ABB RAPID module: CurvedAlign3DP_R7.modx

MODULE CurvedAlign3DP

	VAR jointtarget SDP_0 := [[-4.75, 34.73, 8.1, 0, 47.17, -94.75], [9E9, 9E9, 9E9, 9E9, 9E9, 9E9]];
	VAR jointtarget SDP_1 := [[-3.57, 34.64, 8.25, 0, 47.11, -93.57], [9E9, 9E9, 9E9, 9E9, 9E9, 9E9]];
	VAR jointtarget SDP_2 := [[-2.38, 34.58, 8.36, 0, 47.06, -92.38], [9E9, 9E9, 9E9, 9E9, 9E9, 9E9]];
	VAR jointtarget SDP_3 := [[-1.19, 34.54, 8.43, 0, 47.03, -91.19], [9E9, 9E9, 9E9, 9E9, 9E9, 9E9]];
	VAR jointtarget SDP_4 := [[0, 34.52, 8.45, 0, 47.02, -90], [9E9, 9E9, 9E9, 9E9, 9E9, 9E9]];
	VAR jointtarget SDP_5 := [[1.19, 34.54, 8.43, 0, 47.03, -88.81], [9E9, 9E9, 9E9, 9E9, 9E9, 9E9]];
	VAR jointtarget SDP_6 := [[2.38, 34.58, 8.36, 0, 47.06, -87.62], [9E9, 9E9, 9E9, 9E9, 9E9, 9E9]];
	VAR jointtarget SDP_7 := [[3.57, 34.64, 8.25, 0, 47.11, -86.43], [9E9, 9E9, 9E9, 9E9, 9E9, 9E9]];
	VAR jointtarget SDP_8 := [[4.75, 34.73, 8.1, 0, 47.17, -85.25], [9E9, 9E9, 9E9, 9E9, 9E9, 9E9]];
	VAR jointtarget SDP_9 := [[5.93, 34.85, 7.9, 0, 47.25, -84.07], [9E9, 9E9, 9E9, 9E9, 9E9, 9E9]];
	VAR jointtarget SDP_10 := [[6.27, 34.91, 7.79, 0, 47.3, -79.23], [9E9, 9E9, 9E9, 9E9, 9E9, 9E9]];
	VAR jointtarget SDP_11 := [[6.6, 35.04, 7.57, 0, 47.39, -69.9], [9E9, 9E9, 9E9, 9E9, 9E9, 9E9]];
	VAR jointtarget SDP_12 := [[6.9, 35.22, 7.27, 0, 47.51, -60.6], [9E9, 9E9, 9E9, 9E9, 9E9, 9E9]];
	VAR jointtarget SDP_13 := [[7.17, 35.45, 6.88, 0, 47.68, -51.33], [9E9, 9E9, 9E9, 9E9, 9E9, 9E9]];
	VAR jointtarget SDP_14 := [[7.4, 35.72, 6.41, 0, 47.87, -42.1], [9E9, 9E9, 9E9, 9E9, 9E9, 9E9]];
	VAR jointtarget SDP_15 := [[7.59, 36.03, 5.88, 0, 48.09, -32.91], [9E9, 9E9, 9E9, 9E9, 9E9, 9E9]];
	VAR jointtarget SDP_16 := [[7.73, 36.37, 5.3, 0, 48.34, -23.77], [9E9, 9E9, 9E9, 9E9, 9E9, 9E9]];
	VAR jointtarget SDP_17 := [[7.82, 36.73, 4.68, 0, 48.59, -14.68], [9E9, 9E9, 9E9, 9E9, 9E9, 9E9]];
	VAR jointtarget SDP_18 := [[7.85, 37.1, 4.04, 0, 48.86, -5.65], [9E9, 9E9, 9E9, 9E9, 9E9, 9E9]];
	VAR jointtarget SDP_19 := [[7.83, 37.47, 3.39, 0, 49.13, 3.33], [9E9, 9E9, 9E9, 9E9, 9E9, 9E9]];
	VAR jointtarget SDP_20 := [[7.68, 38.72, 1.22, 0, 50.05, 7.68], [9E9, 9E9, 9E9, 9E9, 9E9, 9E9]];
	VAR jointtarget SDP_21 := [[7.54, 39.99, -0.99, 0, 51, 7.54], [9E9, 9E9, 9E9, 9E9, 9E9, 9E9]];
	VAR jointtarget SDP_22 := [[7.4, 41.28, -3.25, 0, 51.98, 7.4], [9E9, 9E9, 9E9, 9E9, 9E9, 9E9]];
	VAR jointtarget SDP_23 := [[7.26, 42.59, -5.57, 0, 52.98, 7.26], [9E9, 9E9, 9E9, 9E9, 9E9, 9E9]];
	VAR jointtarget SDP_24 := [[7.13, 43.92, -7.93, 0, 54.01, 7.13], [9E9, 9E9, 9E9, 9E9, 9E9, 9E9]];
	VAR jointtarget SDP_25 := [[7.01, 45.28, -10.36, 0, 55.08, 7.01], [9E9, 9E9, 9E9, 9E9, 9E9, 9E9]];
	VAR jointtarget SDP_26 := [[6.89, 46.67, -12.86, 0, 56.19, 6.89], [9E9, 9E9, 9E9, 9E9, 9E9, 9E9]];
	VAR jointtarget SDP_27 := [[6.77, 48.09, -15.43, 0, 57.33, 6.77], [9E9, 9E9, 9E9, 9E9, 9E9, 9E9]];
	VAR jointtarget SDP_28 := [[6.66, 49.56, -18.07, 0, 58.52, 6.66], [9E9, 9E9, 9E9, 9E9, 9E9, 9E9]];
	VAR jointtarget SDP_29 := [[6.55, 51.06, -20.82, 0, 59.75, 6.55], [9E9, 9E9, 9E9, 9E9, 9E9, 9E9]];
	VAR jointtarget SDP_30 := [[6.55, 51.11, -20.9, 0, 59.79, 5.89], [9E9, 9E9, 9E9, 9E9, 9E9, 9E9]];
	VAR jointtarget SDP_31 := [[6.55, 51.15, -20.98, 0, 59.83, 4.56], [9E9, 9E9, 9E9, 9E9, 9E9, 9E9]];
	VAR jointtarget SDP_32 := [[6.55, 51.2, -21.06, 0, 59.87, 3.24], [9E9, 9E9, 9E9, 9E9, 9E9, 9E9]];
	VAR jointtarget SDP_33 := [[6.54, 51.24, -21.14, 0, 59.9, 1.91], [9E9, 9E9, 9E9, 9E9, 9E9, 9E9]];
	VAR jointtarget SDP_34 := [[6.54, 51.29, -21.23, 0, 59.94, 0.59], [9E9, 9E9, 9E9, 9E9, 9E9, 9E9]];
	VAR jointtarget SDP_35 := [[6.54, 51.33, -21.31, 0, 59.98, -0.74], [9E9, 9E9, 9E9, 9E9, 9E9, 9E9]];
	VAR jointtarget SDP_36 := [[6.55, 51.38, -21.39, 0, 60.01, -2.06], [9E9, 9E9, 9E9, 9E9, 9E9, 9E9]];
	VAR jointtarget SDP_37 := [[6.55, 51.42, -21.48, 0, 60.05, -3.38], [9E9, 9E9, 9E9, 9E9, 9E9, 9E9]];
	VAR jointtarget SDP_38 := [[6.55, 51.47, -21.56, 0, 60.09, -4.7], [9E9, 9E9, 9E9, 9E9, 9E9, 9E9]];
	VAR jointtarget SDP_39 := [[6.55, 51.51, -21.64, 0, 60.13, -6.03], [9E9, 9E9, 9E9, 9E9, 9E9, 9E9]];
	VAR jointtarget SDP_40 := [[6.57, 51.7, -21.98, 0, 60.28, -6.68], [9E9, 9E9, 9E9, 9E9, 9E9, 9E9]];
	VAR jointtarget SDP_41 := [[6.58, 51.88, -22.31, 0, 60.43, -6.66], [9E9, 9E9, 9E9, 9E9, 9E9, 9E9]];
	VAR jointtarget SDP_42 := [[6.59, 52.06, -22.65, 0, 60.58, -6.65], [9E9, 9E9, 9E9, 9E9, 9E9, 9E9]];
	VAR jointtarget SDP_43 := [[6.6, 52.25, -22.99, 0, 60.74, -6.64], [9E9, 9E9, 9E9, 9E9, 9E9, 9E9]];
	VAR jointtarget SDP_44 := [[6.62, 52.44, -23.33, 0, 60.89, -6.62], [9E9, 9E9, 9E9, 9E9, 9E9, 9E9]];
	VAR jointtarget SDP_45 := [[6.63, 52.62, -23.67, 0, 61.05, -6.61], [9E9, 9E9, 9E9, 9E9, 9E9, 9E9]];
	VAR jointtarget SDP_46 := [[6.64, 52.81, -24.01, 0, 61.2, -6.6], [9E9, 9E9, 9E9, 9E9, 9E9, 9E9]];
	VAR jointtarget SDP_47 := [[6.65, 53, -24.36, 0, 61.36, -6.59], [9E9, 9E9, 9E9, 9E9, 9E9, 9E9]];
	VAR jointtarget SDP_48 := [[6.67, 53.19, -24.7, 0, 61.52, -6.57], [9E9, 9E9, 9E9, 9E9, 9E9, 9E9]];
	VAR jointtarget SDP_49 := [[6.68, 53.38, -25.05, 0, 61.68, -6.56], [9E9, 9E9, 9E9, 9E9, 9E9, 9E9]];
	VAR jointtarget SDP_50 := [[6.66, 53.75, -25.74, 0, 61.99, 3.75], [9E9, 9E9, 9E9, 9E9, 9E9, 9E9]];
	VAR jointtarget SDP_51 := [[6.58, 54.09, -26.37, 0, 62.27, 24.31], [9E9, 9E9, 9E9, 9E9, 9E9, 9E9]];
	VAR jointtarget SDP_52 := [[6.43, 54.36, -26.86, 0, 62.5, 44.81], [9E9, 9E9, 9E9, 9E9, 9E9, 9E9]];
	VAR jointtarget SDP_53 := [[6.24, 54.52, -27.15, 0, 62.63, 65.27], [9E9, 9E9, 9E9, 9E9, 9E9, 9E9]];
	VAR jointtarget SDP_54 := [[6.04, 54.55, -27.2, 0, 62.66, 85.71], [9E9, 9E9, 9E9, 9E9, 9E9, 9E9]];
	VAR jointtarget SDP_55 := [[5.84, 54.44, -27.01, 0, 62.57, 106.16], [9E9, 9E9, 9E9, 9E9, 9E9, 9E9]];
	VAR jointtarget SDP_56 := [[5.67, 54.21, -26.59, 0, 62.38, 126.64], [9E9, 9E9, 9E9, 9E9, 9E9, 9E9]];
	VAR jointtarget SDP_57 := [[5.56, 53.89, -26, 0, 62.11, 147.18], [9E9, 9E9, 9E9, 9E9, 9E9, 9E9]];
	VAR jointtarget SDP_58 := [[5.52, 53.53, -25.33, 0, 61.8, 167.78], [9E9, 9E9, 9E9, 9E9, 9E9, 9E9]];
	VAR jointtarget SDP_59 := [[5.55, 53.16, -24.66, 0, 61.5, 188.46], [9E9, 9E9, 9E9, 9E9, 9E9, 9E9]];
	VAR jointtarget SDP_60 := [[5.58, 52.98, -24.33, 0, 61.35, 198.82], [9E9, 9E9, 9E9, 9E9, 9E9, 9E9]];
	VAR jointtarget SDP_61 := [[5.62, 52.8, -24, 0, 61.2, 198.86], [9E9, 9E9, 9E9, 9E9, 9E9, 9E9]];
	VAR jointtarget SDP_62 := [[5.65, 52.62, -23.67, 0, 61.05, 198.89], [9E9, 9E9, 9E9, 9E9, 9E9, 9E9]];
	VAR jointtarget SDP_63 := [[5.69, 52.45, -23.35, 0, 60.9, 198.93], [9E9, 9E9, 9E9, 9E9, 9E9, 9E9]];
	VAR jointtarget SDP_64 := [[5.72, 52.27, -23.02, 0, 60.75, 198.96], [9E9, 9E9, 9E9, 9E9, 9E9, 9E9]];
	VAR jointtarget SDP_65 := [[5.76, 52.09, -22.7, 0, 60.61, 199], [9E9, 9E9, 9E9, 9E9, 9E9, 9E9]];
	VAR jointtarget SDP_66 := [[5.79, 51.92, -22.38, 0, 60.46, 199.03], [9E9, 9E9, 9E9, 9E9, 9E9, 9E9]];
	VAR jointtarget SDP_67 := [[5.83, 51.74, -22.06, 0, 60.32, 199.07], [9E9, 9E9, 9E9, 9E9, 9E9, 9E9]];
	VAR jointtarget SDP_68 := [[5.87, 51.57, -21.74, 0, 60.17, 199.11], [9E9, 9E9, 9E9, 9E9, 9E9, 9E9]];
	VAR jointtarget SDP_69 := [[5.9, 51.4, -21.43, 0, 60.03, 199.14], [9E9, 9E9, 9E9, 9E9, 9E9, 9E9]];
	VAR jointtarget SDP_70 := [[5.91, 51.35, -21.35, 0, 59.99, 198.49], [9E9, 9E9, 9E9, 9E9, 9E9, 9E9]];
	VAR jointtarget SDP_71 := [[5.92, 51.31, -21.27, 0, 59.96, 197.17], [9E9, 9E9, 9E9, 9E9, 9E9, 9E9]];
	VAR jointtarget SDP_72 := [[5.93, 51.27, -21.19, 0, 59.92, 195.86], [9E9, 9E9, 9E9, 9E9, 9E9, 9E9]];
	VAR jointtarget SDP_73 := [[5.93, 51.22, -21.11, 0, 59.89, 194.54], [9E9, 9E9, 9E9, 9E9, 9E9, 9E9]];
	VAR jointtarget SDP_74 := [[5.94, 51.18, -21.03, 0, 59.85, 193.22], [9E9, 9E9, 9E9, 9E9, 9E9, 9E9]];
	VAR jointtarget SDP_75 := [[5.94, 51.13, -20.95, 0, 59.81, 191.9], [9E9, 9E9, 9E9, 9E9, 9E9, 9E9]];
	VAR jointtarget SDP_76 := [[5.95, 51.09, -20.87, 0, 59.78, 190.58], [9E9, 9E9, 9E9, 9E9, 9E9, 9E9]];
	VAR jointtarget SDP_77 := [[5.95, 51.04, -20.78, 0, 59.74, 189.26], [9E9, 9E9, 9E9, 9E9, 9E9, 9E9]];
	VAR jointtarget SDP_78 := [[5.96, 51, -20.7, 0, 59.7, 187.94], [9E9, 9E9, 9E9, 9E9, 9E9, 9E9]];
	VAR jointtarget SDP_79 := [[5.96, 50.96, -20.62, 0, 59.67, 186.62], [9E9, 9E9, 9E9, 9E9, 9E9, 9E9]];
	VAR jointtarget SDP_80 := [[6.05, 49.55, -18.06, 0, 58.51, 186.05], [9E9, 9E9, 9E9, 9E9, 9E9, 9E9]];
	VAR jointtarget SDP_81 := [[6.15, 48.17, -15.57, 0, 57.4, 186.15], [9E9, 9E9, 9E9, 9E9, 9E9, 9E9]];
	VAR jointtarget SDP_82 := [[6.25, 46.84, -13.15, 0, 56.32, 186.25], [9E9, 9E9, 9E9, 9E9, 9E9, 9E9]];
	VAR jointtarget SDP_83 := [[6.35, 45.53, -10.81, 0, 55.28, 186.35], [9E9, 9E9, 9E9, 9E9, 9E9, 9E9]];
	VAR jointtarget SDP_84 := [[6.46, 44.25, -8.52, 0, 54.27, 186.46], [9E9, 9E9, 9E9, 9E9, 9E9, 9E9]];
	VAR jointtarget SDP_85 := [[6.56, 42.99, -6.28, 0, 53.29, 186.56], [9E9, 9E9, 9E9, 9E9, 9E9, 9E9]];
	VAR jointtarget SDP_86 := [[6.68, 41.76, -4.09, 0, 52.34, 186.68], [9E9, 9E9, 9E9, 9E9, 9E9, 9E9]];
	VAR jointtarget SDP_87 := [[6.79, 40.54, -1.95, 0, 51.41, 186.79], [9E9, 9E9, 9E9, 9E9, 9E9, 9E9]];
	VAR jointtarget SDP_88 := [[6.91, 39.34, 0.14, 0, 50.52, 186.91], [9E9, 9E9, 9E9, 9E9, 9E9, 9E9]];
	VAR jointtarget SDP_89 := [[7.04, 38.16, 2.2, 0, 49.64, 187.04], [9E9, 9E9, 9E9, 9E9, 9E9, 9E9]];
	VAR jointtarget SDP_90 := [[7.05, 37.78, 2.85, 0, 49.36, 182.55], [9E9, 9E9, 9E9, 9E9, 9E9, 9E9]];
	VAR jointtarget SDP_91 := [[7.02, 37.41, 3.5, 0, 49.09, 173.52], [9E9, 9E9, 9E9, 9E9, 9E9, 9E9]];
	VAR jointtarget SDP_92 := [[6.93, 37.05, 4.12, 0, 48.83, 164.43], [9E9, 9E9, 9E9, 9E9, 9E9, 9E9]];
	VAR jointtarget SDP_93 := [[6.78, 36.71, 4.7, 0, 48.58, 155.28], [9E9, 9E9, 9E9, 9E9, 9E9, 9E9]];
	VAR jointtarget SDP_94 := [[6.6, 36.4, 5.23, 0, 48.36, 146.1], [9E9, 9E9, 9E9, 9E9, 9E9, 9E9]];
	VAR jointtarget SDP_95 := [[6.36, 36.13, 5.7, 0, 48.17, 136.86], [9E9, 9E9, 9E9, 9E9, 9E9, 9E9]];
	VAR jointtarget SDP_96 := [[6.09, 35.91, 6.09, 0, 48, 127.59], [9E9, 9E9, 9E9, 9E9, 9E9, 9E9]];
	VAR jointtarget SDP_97 := [[5.79, 35.73, 6.39, 0, 47.88, 118.29], [9E9, 9E9, 9E9, 9E9, 9E9, 9E9]];
	VAR jointtarget SDP_98 := [[5.47, 35.61, 6.6, 0, 47.79, 108.97], [9E9, 9E9, 9E9, 9E9, 9E9, 9E9]];
	VAR jointtarget SDP_99 := [[5.13, 35.55, 6.7, 0, 47.75, 99.63], [9E9, 9E9, 9E9, 9E9, 9E9, 9E9]];
	VAR jointtarget SDP_100 := [[4.07, 35.46, 6.86, 0, 47.68, 94.07], [9E9, 9E9, 9E9, 9E9, 9E9, 9E9]];
	VAR jointtarget SDP_101 := [[3.01, 35.39, 6.98, 0, 47.63, 93.01], [9E9, 9E9, 9E9, 9E9, 9E9, 9E9]];
	VAR jointtarget SDP_102 := [[1.95, 35.34, 7.06, 0, 47.6, 91.95], [9E9, 9E9, 9E9, 9E9, 9E9, 9E9]];
	VAR jointtarget SDP_103 := [[0.89, 35.31, 7.11, 0, 47.58, 90.89], [9E9, 9E9, 9E9, 9E9, 9E9, 9E9]];
	VAR jointtarget SDP_104 := [[-0.18, 35.3, 7.12, 0, 47.57, 89.82], [9E9, 9E9, 9E9, 9E9, 9E9, 9E9]];
	VAR jointtarget SDP_105 := [[-1.24, 35.32, 7.1, 0, 47.58, 88.76], [9E9, 9E9, 9E9, 9E9, 9E9, 9E9]];
	VAR jointtarget SDP_106 := [[-2.31, 35.35, 7.04, 0, 47.61, 87.69], [9E9, 9E9, 9E9, 9E9, 9E9, 9E9]];
	VAR jointtarget SDP_107 := [[-3.37, 35.41, 6.94, 0, 47.65, 86.63], [9E9, 9E9, 9E9, 9E9, 9E9, 9E9]];
	VAR jointtarget SDP_108 := [[-4.43, 35.48, 6.81, 0, 47.7, 85.57], [9E9, 9E9, 9E9, 9E9, 9E9, 9E9]];
	VAR jointtarget SDP_109 := [[-5.48, 35.58, 6.64, 0, 47.77, 84.52], [9E9, 9E9, 9E9, 9E9, 9E9, 9E9]];
	VAR jointtarget SDP_110 := [[-5.59, 35.59, 6.63, 0, 47.78, 86.6], [9E9, 9E9, 9E9, 9E9, 9E9, 9E9]];
	VAR jointtarget SDP_111 := [[-5.71, 35.59, 6.64, 0, 47.78, 90.88], [9E9, 9E9, 9E9, 9E9, 9E9, 9E9]];
	VAR jointtarget SDP_112 := [[-5.82, 35.58, 6.65, 0, 47.77, 95.15], [9E9, 9E9, 9E9, 9E9, 9E9, 9E9]];
	VAR jointtarget SDP_113 := [[-5.93, 35.56, 6.69, 0, 47.75, 99.43], [9E9, 9E9, 9E9, 9E9, 9E9, 9E9]];
	VAR jointtarget SDP_114 := [[-6.04, 35.53, 6.74, 0, 47.73, 103.71], [9E9, 9E9, 9E9, 9E9, 9E9, 9E9]];
	VAR jointtarget SDP_115 := [[-6.14, 35.49, 6.8, 0, 47.71, 107.99], [9E9, 9E9, 9E9, 9E9, 9E9, 9E9]];
	VAR jointtarget SDP_116 := [[-6.25, 35.45, 6.88, 0, 47.68, 112.27], [9E9, 9E9, 9E9, 9E9, 9E9, 9E9]];
	VAR jointtarget SDP_117 := [[-6.35, 35.39, 6.97, 0, 47.64, 116.56], [9E9, 9E9, 9E9, 9E9, 9E9, 9E9]];
	VAR jointtarget SDP_118 := [[-6.44, 35.33, 7.08, 0, 47.59, 120.85], [9E9, 9E9, 9E9, 9E9, 9E9, 9E9]];
	VAR jointtarget SDP_119 := [[-6.54, 35.26, 7.19, 0, 47.54, 125.15], [9E9, 9E9, 9E9, 9E9, 9E9, 9E9]];
	VAR jointtarget SDP_120 := [[-6.59, 35.22, 7.27, 0, 47.51, 127.29], [9E9, 9E9, 9E9, 9E9, 9E9, 9E9]];
	VAR jointtarget SDP_121 := [[-6.64, 35.17, 7.34, 0, 47.48, 127.23], [9E9, 9E9, 9E9, 9E9, 9E9, 9E9]];
	VAR jointtarget SDP_122 := [[-6.7, 35.13, 7.42, 0, 47.45, 127.18], [9E9, 9E9, 9E9, 9E9, 9E9, 9E9]];
	VAR jointtarget SDP_123 := [[-6.75, 35.09, 7.49, 0, 47.42, 127.12], [9E9, 9E9, 9E9, 9E9, 9E9, 9E9]];
	VAR jointtarget SDP_124 := [[-6.81, 35.04, 7.57, 0, 47.39, 127.07], [9E9, 9E9, 9E9, 9E9, 9E9, 9E9]];
	VAR jointtarget SDP_125 := [[-6.86, 35, 7.64, 0, 47.36, 127.01], [9E9, 9E9, 9E9, 9E9, 9E9, 9E9]];
	VAR jointtarget SDP_126 := [[-6.92, 34.96, 7.71, 0, 47.33, 126.96], [9E9, 9E9, 9E9, 9E9, 9E9, 9E9]];
	VAR jointtarget SDP_127 := [[-6.97, 34.91, 7.79, 0, 47.3, 126.91], [9E9, 9E9, 9E9, 9E9, 9E9, 9E9]];
	VAR jointtarget SDP_128 := [[-7.03, 34.87, 7.86, 0, 47.27, 126.85], [9E9, 9E9, 9E9, 9E9, 9E9, 9E9]];
	VAR jointtarget SDP_129 := [[-7.08, 34.83, 7.94, 0, 47.24, 126.8], [9E9, 9E9, 9E9, 9E9, 9E9, 9E9]];
	VAR jointtarget SDP_130 := [[-7.39, 34.69, 8.17, 0, 47.14, 113.1], [9E9, 9E9, 9E9, 9E9, 9E9, 9E9]];
	VAR jointtarget SDP_131 := [[-7.72, 34.71, 8.13, 0, 47.16, 85.99], [9E9, 9E9, 9E9, 9E9, 9E9, 9E9]];
	VAR jointtarget SDP_132 := [[-8.01, 34.89, 7.82, 0, 47.28, 58.93], [9E9, 9E9, 9E9, 9E9, 9E9, 9E9]];
	VAR jointtarget SDP_133 := [[-8.18, 35.19, 7.32, 0, 47.49, 31.98], [9E9, 9E9, 9E9, 9E9, 9E9, 9E9]];
	VAR jointtarget SDP_134 := [[-8.21, 35.54, 6.72, 0, 47.74, 5.18], [9E9, 9E9, 9E9, 9E9, 9E9, 9E9]];
	VAR jointtarget SDP_135 := [[-8.09, 35.87, 6.16, 0, 47.98, -21.48], [9E9, 9E9, 9E9, 9E9, 9E9, 9E9]];
	VAR jointtarget SDP_136 := [[-7.85, 36.1, 5.75, 0, 48.14, -48.01], [9E9, 9E9, 9E9, 9E9, 9E9, 9E9]];
	VAR jointtarget SDP_137 := [[-7.53, 36.2, 5.59, 0, 48.21, -74.47], [9E9, 9E9, 9E9, 9E9, 9E9, 9E9]];
	VAR jointtarget SDP_138 := [[-7.21, 36.13, 5.71, 0, 48.16, -100.93], [9E9, 9E9, 9E9, 9E9, 9E9, 9E9]];
	VAR jointtarget SDP_139 := [[-6.96, 35.91, 6.08, 0, 48.01, -127.44], [9E9, 9E9, 9E9, 9E9, 9E9, 9E9]];
	VAR jointtarget SDP_140 := [[-6.9, 35.84, 6.2, 0, 47.96, -140.78], [9E9, 9E9, 9E9, 9E9, 9E9, 9E9]];
	VAR jointtarget SDP_141 := [[-6.85, 35.77, 6.32, 0, 47.91, -140.72], [9E9, 9E9, 9E9, 9E9, 9E9, 9E9]];
	VAR jointtarget SDP_142 := [[-6.79, 35.7, 6.45, 0, 47.86, -140.67], [9E9, 9E9, 9E9, 9E9, 9E9, 9E9]];
	VAR jointtarget SDP_143 := [[-6.74, 35.63, 6.57, 0, 47.81, -140.62], [9E9, 9E9, 9E9, 9E9, 9E9, 9E9]];
	VAR jointtarget SDP_144 := [[-6.68, 35.56, 6.69, 0, 47.75, -140.56], [9E9, 9E9, 9E9, 9E9, 9E9, 9E9]];
	VAR jointtarget SDP_145 := [[-6.63, 35.49, 6.81, 0, 47.7, -140.51], [9E9, 9E9, 9E9, 9E9, 9E9, 9E9]];
	VAR jointtarget SDP_146 := [[-6.58, 35.42, 6.93, 0, 47.65, -140.45], [9E9, 9E9, 9E9, 9E9, 9E9, 9E9]];
	VAR jointtarget SDP_147 := [[-6.52, 35.34, 7.05, 0, 47.6, -140.4], [9E9, 9E9, 9E9, 9E9, 9E9, 9E9]];
	VAR jointtarget SDP_148 := [[-6.47, 35.27, 7.17, 0, 47.55, -140.34], [9E9, 9E9, 9E9, 9E9, 9E9, 9E9]];
	VAR jointtarget SDP_149 := [[-6.41, 35.2, 7.29, 0, 47.5, -140.29], [9E9, 9E9, 9E9, 9E9, 9E9, 9E9]];
	VAR jointtarget SDP_150 := [[-6.38, 35.17, 7.35, 0, 47.48, -139.16], [9E9, 9E9, 9E9, 9E9, 9E9, 9E9]];
	VAR jointtarget SDP_151 := [[-6.36, 35.14, 7.4, 0, 47.46, -136.92], [9E9, 9E9, 9E9, 9E9, 9E9, 9E9]];
	VAR jointtarget SDP_152 := [[-6.33, 35.11, 7.45, 0, 47.44, -134.69], [9E9, 9E9, 9E9, 9E9, 9E9, 9E9]];
	VAR jointtarget SDP_153 := [[-6.3, 35.08, 7.5, 0, 47.42, -132.45], [9E9, 9E9, 9E9, 9E9, 9E9, 9E9]];
	VAR jointtarget SDP_154 := [[-6.27, 35.06, 7.54, 0, 47.4, -130.22], [9E9, 9E9, 9E9, 9E9, 9E9, 9E9]];
	VAR jointtarget SDP_155 := [[-6.24, 35.03, 7.58, 0, 47.39, -127.98], [9E9, 9E9, 9E9, 9E9, 9E9, 9E9]];
	VAR jointtarget SDP_156 := [[-6.21, 35.01, 7.63, 0, 47.37, -125.74], [9E9, 9E9, 9E9, 9E9, 9E9, 9E9]];
	VAR jointtarget SDP_157 := [[-6.18, 34.98, 7.66, 0, 47.35, -123.5], [9E9, 9E9, 9E9, 9E9, 9E9, 9E9]];
	VAR jointtarget SDP_158 := [[-6.14, 34.96, 7.7, 0, 47.34, -121.26], [9E9, 9E9, 9E9, 9E9, 9E9, 9E9]];
	VAR jointtarget SDP_159 := [[-6.11, 34.94, 7.74, 0, 47.33, -119.01], [9E9, 9E9, 9E9, 9E9, 9E9, 9E9]];
	VAR jointtarget SDP_160 := [[-6.09, 34.93, 7.75, 0, 47.32, -117.89], [9E9, 9E9, 9E9, 9E9, 9E9, 9E9]];
	VAR jointtarget SDP_161 := [[-6.07, 34.92, 7.77, 0, 47.32, -117.87], [9E9, 9E9, 9E9, 9E9, 9E9, 9E9]];
	VAR jointtarget SDP_162 := [[-6.05, 34.91, 7.78, 0, 47.31, -117.86], [9E9, 9E9, 9E9, 9E9, 9E9, 9E9]];
	VAR jointtarget SDP_163 := [[-6.04, 34.9, 7.8, 0, 47.3, -117.84], [9E9, 9E9, 9E9, 9E9, 9E9, 9E9]];
	VAR jointtarget SDP_164 := [[-6.02, 34.88, 7.82, 0, 47.3, -117.82], [9E9, 9E9, 9E9, 9E9, 9E9, 9E9]];
	VAR jointtarget SDP_165 := [[-6, 34.87, 7.83, 0, 47.29, -117.8], [9E9, 9E9, 9E9, 9E9, 9E9, 9E9]];
	VAR jointtarget SDP_166 := [[-5.98, 34.86, 7.85, 0, 47.28, -117.79], [9E9, 9E9, 9E9, 9E9, 9E9, 9E9]];
	VAR jointtarget SDP_167 := [[-5.97, 34.85, 7.87, 0, 47.28, -117.77], [9E9, 9E9, 9E9, 9E9, 9E9, 9E9]];
	VAR jointtarget SDP_168 := [[-5.95, 34.84, 7.88, 0, 47.27, -117.75], [9E9, 9E9, 9E9, 9E9, 9E9, 9E9]];
	VAR jointtarget SDP_169 := [[-5.93, 34.83, 7.9, 0, 47.27, -117.73], [9E9, 9E9, 9E9, 9E9, 9E9, 9E9]];
	VAR jointtarget SDP_170 := [[-4.75, 34.72, 8.1, 0, 47.19, -94.75], [9E9, 9E9, 9E9, 9E9, 9E9, 9E9]];
	VAR jointtarget SDP_171 := [[-3.57, 34.63, 8.25, 0, 47.12, -93.57], [9E9, 9E9, 9E9, 9E9, 9E9, 9E9]];
	VAR jointtarget SDP_172 := [[-2.38, 34.56, 8.36, 0, 47.08, -92.38], [9E9, 9E9, 9E9, 9E9, 9E9, 9E9]];
	VAR jointtarget SDP_173 := [[-1.19, 34.52, 8.43, 0, 47.05, -91.19], [9E9, 9E9, 9E9, 9E9, 9E9, 9E9]];
	VAR jointtarget SDP_174 := [[0, 34.51, 8.45, 0, 47.04, -90], [9E9, 9E9, 9E9, 9E9, 9E9, 9E9]];
	VAR jointtarget SDP_175 := [[1.19, 34.52, 8.43, 0, 47.05, -88.81], [9E9, 9E9, 9E9, 9E9, 9E9, 9E9]];
	VAR jointtarget SDP_176 := [[2.38, 34.56, 8.36, 0, 47.08, -87.62], [9E9, 9E9, 9E9, 9E9, 9E9, 9E9]];
	VAR jointtarget SDP_177 := [[3.57, 34.63, 8.25, 0, 47.12, -86.43], [9E9, 9E9, 9E9, 9E9, 9E9, 9E9]];
	VAR jointtarget SDP_178 := [[4.75, 34.72, 8.1, 0, 47.19, -85.25], [9E9, 9E9, 9E9, 9E9, 9E9, 9E9]];
	VAR jointtarget SDP_179 := [[5.93, 34.83, 7.9, 0, 47.27, -84.07], [9E9, 9E9, 9E9, 9E9, 9E9, 9E9]];
	VAR jointtarget SDP_180 := [[6.27, 34.9, 7.79, 0, 47.31, -79.23], [9E9, 9E9, 9E9, 9E9, 9E9, 9E9]];
	VAR jointtarget SDP_181 := [[6.6, 35.03, 7.57, 0, 47.4, -69.9], [9E9, 9E9, 9E9, 9E9, 9E9, 9E9]];
	VAR jointtarget SDP_182 := [[6.9, 35.2, 7.27, 0, 47.53, -60.6], [9E9, 9E9, 9E9, 9E9, 9E9, 9E9]];
	VAR jointtarget SDP_183 := [[7.17, 35.43, 6.87, 0, 47.69, -51.33], [9E9, 9E9, 9E9, 9E9, 9E9, 9E9]];
	VAR jointtarget SDP_184 := [[7.4, 35.71, 6.41, 0, 47.89, -42.1], [9E9, 9E9, 9E9, 9E9, 9E9, 9E9]];
	VAR jointtarget SDP_185 := [[7.59, 36.02, 5.88, 0, 48.11, -32.91], [9E9, 9E9, 9E9, 9E9, 9E9, 9E9]];
	VAR jointtarget SDP_186 := [[7.73, 36.36, 5.29, 0, 48.35, -23.77], [9E9, 9E9, 9E9, 9E9, 9E9, 9E9]];
	VAR jointtarget SDP_187 := [[7.82, 36.71, 4.68, 0, 48.61, -14.68], [9E9, 9E9, 9E9, 9E9, 9E9, 9E9]];
	VAR jointtarget SDP_188 := [[7.85, 37.09, 4.04, 0, 48.88, -5.65], [9E9, 9E9, 9E9, 9E9, 9E9, 9E9]];
	VAR jointtarget SDP_189 := [[7.83, 37.46, 3.39, 0, 49.15, 3.33], [9E9, 9E9, 9E9, 9E9, 9E9, 9E9]];
	VAR jointtarget SDP_190 := [[7.68, 38.69, 1.26, 0, 50.05, 7.68], [9E9, 9E9, 9E9, 9E9, 9E9, 9E9]];
	VAR jointtarget SDP_191 := [[7.54, 39.93, -0.92, 0, 50.98, 7.54], [9E9, 9E9, 9E9, 9E9, 9E9, 9E9]];
	VAR jointtarget SDP_192 := [[7.4, 41.2, -3.13, 0, 51.94, 7.4], [9E9, 9E9, 9E9, 9E9, 9E9, 9E9]];
	VAR jointtarget SDP_193 := [[7.27, 42.48, -5.4, 0, 52.92, 7.27], [9E9, 9E9, 9E9, 9E9, 9E9, 9E9]];
	VAR jointtarget SDP_194 := [[7.15, 43.79, -7.72, 0, 53.93, 7.15], [9E9, 9E9, 9E9, 9E9, 9E9, 9E9]];
	VAR jointtarget SDP_195 := [[7.02, 45.12, -10.1, 0, 54.98, 7.02], [9E9, 9E9, 9E9, 9E9, 9E9, 9E9]];
	VAR jointtarget SDP_196 := [[6.9, 46.48, -12.54, 0, 56.06, 6.9], [9E9, 9E9, 9E9, 9E9, 9E9, 9E9]];
	VAR jointtarget SDP_197 := [[6.79, 47.88, -15.06, 0, 57.18, 6.79], [9E9, 9E9, 9E9, 9E9, 9E9, 9E9]];
	VAR jointtarget SDP_198 := [[6.68, 49.31, -17.65, 0, 58.34, 6.68], [9E9, 9E9, 9E9, 9E9, 9E9, 9E9]];
	VAR jointtarget SDP_199 := [[6.57, 50.78, -20.32, 0, 59.54, 6.57], [9E9, 9E9, 9E9, 9E9, 9E9, 9E9]];
	VAR jointtarget SDP_200 := [[6.56, 50.93, -20.59, 0, 59.66, 8.75], [9E9, 9E9, 9E9, 9E9, 9E9, 9E9]];
	VAR jointtarget SDP_201 := [[6.54, 51.07, -20.85, 0, 59.78, 13.12], [9E9, 9E9, 9E9, 9E9, 9E9, 9E9]];
	VAR jointtarget SDP_202 := [[6.51, 51.21, -21.12, 0, 59.9, 17.48], [9E9, 9E9, 9E9, 9E9, 9E9, 9E9]];
	VAR jointtarget SDP_203 := [[6.48, 51.35, -21.37, 0, 60.02, 21.83], [9E9, 9E9, 9E9, 9E9, 9E9, 9E9]];
	VAR jointtarget SDP_204 := [[6.44, 51.49, -21.62, 0, 60.13, 26.18], [9E9, 9E9, 9E9, 9E9, 9E9, 9E9]];
	VAR jointtarget SDP_205 := [[6.39, 51.62, -21.85, 0, 60.24, 30.52], [9E9, 9E9, 9E9, 9E9, 9E9, 9E9]];
	VAR jointtarget SDP_206 := [[6.34, 51.74, -22.08, 0, 60.34, 34.86], [9E9, 9E9, 9E9, 9E9, 9E9, 9E9]];
	VAR jointtarget SDP_207 := [[6.28, 51.86, -22.3, 0, 60.44, 39.19], [9E9, 9E9, 9E9, 9E9, 9E9, 9E9]];
	VAR jointtarget SDP_208 := [[6.22, 51.97, -22.5, 0, 60.53, 43.51], [9E9, 9E9, 9E9, 9E9, 9E9, 9E9]];
	VAR jointtarget SDP_209 := [[6.15, 52.07, -22.69, 0, 60.61, 47.83], [9E9, 9E9, 9E9, 9E9, 9E9, 9E9]];
	VAR jointtarget SDP_210 := [[6.11, 52.13, -22.8, 0, 60.66, 49.99], [9E9, 9E9, 9E9, 9E9, 9E9, 9E9]];
	VAR jointtarget SDP_211 := [[6.07, 52.19, -22.9, 0, 60.71, 49.95], [9E9, 9E9, 9E9, 9E9, 9E9, 9E9]];
	VAR jointtarget SDP_212 := [[6.03, 52.25, -23.01, 0, 60.76, 49.9], [9E9, 9E9, 9E9, 9E9, 9E9, 9E9]];
	VAR jointtarget SDP_213 := [[5.99, 52.31, -23.12, 0, 60.81, 49.86], [9E9, 9E9, 9E9, 9E9, 9E9, 9E9]];
	VAR jointtarget SDP_214 := [[5.94, 52.37, -23.23, 0, 60.86, 49.82], [9E9, 9E9, 9E9, 9E9, 9E9, 9E9]];
	VAR jointtarget SDP_215 := [[5.9, 52.43, -23.34, 0, 60.91, 49.78], [9E9, 9E9, 9E9, 9E9, 9E9, 9E9]];
	VAR jointtarget SDP_216 := [[5.86, 52.49, -23.45, 0, 60.96, 49.74], [9E9, 9E9, 9E9, 9E9, 9E9, 9E9]];
	VAR jointtarget SDP_217 := [[5.82, 52.55, -23.56, 0, 61.01, 49.7], [9E9, 9E9, 9E9, 9E9, 9E9, 9E9]];
	VAR jointtarget SDP_218 := [[5.78, 52.61, -23.67, 0, 61.06, 49.66], [9E9, 9E9, 9E9, 9E9, 9E9, 9E9]];
	VAR jointtarget SDP_219 := [[5.74, 52.67, -23.79, 0, 61.11, 49.61], [9E9, 9E9, 9E9, 9E9, 9E9, 9E9]];
	VAR jointtarget SDP_220 := [[5.58, 53.04, -24.46, 0, 61.42, 36.07], [9E9, 9E9, 9E9, 9E9, 9E9, 9E9]];
	VAR jointtarget SDP_221 := [[5.54, 53.5, -25.3, 0, 61.8, 9.25], [9E9, 9E9, 9E9, 9E9, 9E9, 9E9]];
	VAR jointtarget SDP_222 := [[5.62, 53.94, -26.11, 0, 62.17, -17.44], [9E9, 9E9, 9E9, 9E9, 9E9, 9E9]];
	VAR jointtarget SDP_223 := [[5.8, 54.28, -26.74, 0, 62.46, -44.04], [9E9, 9E9, 9E9, 9E9, 9E9, 9E9]];
	VAR jointtarget SDP_224 := [[6.04, 54.44, -27.02, 0, 62.59, -70.57], [9E9, 9E9, 9E9, 9E9, 9E9, 9E9]];
	VAR jointtarget SDP_225 := [[6.3, 54.38, -26.91, 0, 62.54, -97.09], [9E9, 9E9, 9E9, 9E9, 9E9, 9E9]];
	VAR jointtarget SDP_226 := [[6.51, 54.12, -26.43, 0, 62.32, -123.65], [9E9, 9E9, 9E9, 9E9, 9E9, 9E9]];
	VAR jointtarget SDP_227 := [[6.64, 53.71, -25.68, 0, 61.97, -150.3], [9E9, 9E9, 9E9, 9E9, 9E9, 9E9]];
	VAR jointtarget SDP_228 := [[6.66, 53.25, -24.83, 0, 61.59, -177.06], [9E9, 9E9, 9E9, 9E9, 9E9, 9E9]];
	VAR jointtarget SDP_229 := [[6.55, 52.83, -24.06, 0, 61.24, -203.94], [9E9, 9E9, 9E9, 9E9, 9E9, 9E9]];
	VAR jointtarget SDP_230 := [[6.52, 52.75, -23.93, 0, 61.18, -217.36], [9E9, 9E9, 9E9, 9E9, 9E9, 9E9]];
	VAR jointtarget SDP_231 := [[6.48, 52.68, -23.79, 0, 61.11, -217.39], [9E9, 9E9, 9E9, 9E9, 9E9, 9E9]];
	VAR jointtarget SDP_232 := [[6.45, 52.6, -23.65, 0, 61.05, -217.42], [9E9, 9E9, 9E9, 9E9, 9E9, 9E9]];
	VAR jointtarget SDP_233 := [[6.42, 52.53, -23.52, 0, 60.99, -217.46], [9E9, 9E9, 9E9, 9E9, 9E9, 9E9]];
	VAR jointtarget SDP_234 := [[6.39, 52.45, -23.38, 0, 60.93, -217.49], [9E9, 9E9, 9E9, 9E9, 9E9, 9E9]];
	VAR jointtarget SDP_235 := [[6.35, 52.38, -23.25, 0, 60.87, -217.52], [9E9, 9E9, 9E9, 9E9, 9E9, 9E9]];
	VAR jointtarget SDP_236 := [[6.32, 52.31, -23.11, 0, 60.81, -217.56], [9E9, 9E9, 9E9, 9E9, 9E9, 9E9]];
	VAR jointtarget SDP_237 := [[6.29, 52.23, -22.98, 0, 60.74, -217.59], [9E9, 9E9, 9E9, 9E9, 9E9, 9E9]];
	VAR jointtarget SDP_238 := [[6.25, 52.16, -22.84, 0, 60.68, -217.62], [9E9, 9E9, 9E9, 9E9, 9E9, 9E9]];
	VAR jointtarget SDP_239 := [[6.22, 52.09, -22.71, 0, 60.62, -217.66], [9E9, 9E9, 9E9, 9E9, 9E9, 9E9]];
	VAR jointtarget SDP_240 := [[6.17, 51.96, -22.48, 0, 60.52, -215.51], [9E9, 9E9, 9E9, 9E9, 9E9, 9E9]];
	VAR jointtarget SDP_241 := [[6.12, 51.83, -22.24, 0, 60.41, -211.17], [9E9, 9E9, 9E9, 9E9, 9E9, 9E9]];
	VAR jointtarget SDP_242 := [[6.08, 51.7, -22, 0, 60.3, -206.83], [9E9, 9E9, 9E9, 9E9, 9E9, 9E9]];
	VAR jointtarget SDP_243 := [[6.05, 51.56, -21.74, 0, 60.18, -202.47], [9E9, 9E9, 9E9, 9E9, 9E9, 9E9]];
	VAR jointtarget SDP_244 := [[6.02, 51.41, -21.48, 0, 60.07, -198.11], [9E9, 9E9, 9E9, 9E9, 9E9, 9E9]];
	VAR jointtarget SDP_245 := [[6, 51.27, -21.21, 0, 59.94, -193.75], [9E9, 9E9, 9E9, 9E9, 9E9, 9E9]];
	VAR jointtarget SDP_246 := [[5.98, 51.12, -20.94, 0, 59.82, -189.38], [9E9, 9E9, 9E9, 9E9, 9E9, 9E9]];
	VAR jointtarget SDP_247 := [[5.97, 50.97, -20.67, 0, 59.7, -185], [9E9, 9E9, 9E9, 9E9, 9E9, 9E9]];
	VAR jointtarget SDP_248 := [[5.97, 50.82, -20.4, 0, 59.58, -180.61], [9E9, 9E9, 9E9, 9E9, 9E9, 9E9]];
	VAR jointtarget SDP_249 := [[5.98, 50.67, -20.13, 0, 59.46, -176.22], [9E9, 9E9, 9E9, 9E9, 9E9, 9E9]];
	VAR jointtarget SDP_250 := [[6.07, 49.3, -17.63, 0, 58.33, -173.93], [9E9, 9E9, 9E9, 9E9, 9E9, 9E9]];
	VAR jointtarget SDP_251 := [[6.16, 47.96, -15.2, 0, 57.24, -173.84], [9E9, 9E9, 9E9, 9E9, 9E9, 9E9]];
	VAR jointtarget SDP_252 := [[6.26, 46.65, -12.84, 0, 56.19, -173.74], [9E9, 9E9, 9E9, 9E9, 9E9, 9E9]];
	VAR jointtarget SDP_253 := [[6.36, 45.37, -10.54, 0, 55.17, -173.64], [9E9, 9E9, 9E9, 9E9, 9E9, 9E9]];
	VAR jointtarget SDP_254 := [[6.47, 44.11, -8.3, 0, 54.19, -173.53], [9E9, 9E9, 9E9, 9E9, 9E9, 9E9]];
	VAR jointtarget SDP_255 := [[6.57, 42.88, -6.11, 0, 53.23, -173.43], [9E9, 9E9, 9E9, 9E9, 9E9, 9E9]];
	VAR jointtarget SDP_256 := [[6.68, 41.67, -3.97, 0, 52.3, -173.32], [9E9, 9E9, 9E9, 9E9, 9E9, 9E9]];
	VAR jointtarget SDP_257 := [[6.8, 40.48, -1.88, 0, 51.39, -173.2], [9E9, 9E9, 9E9, 9E9, 9E9, 9E9]];
	VAR jointtarget SDP_258 := [[6.92, 39.31, 0.18, 0, 50.51, -173.08], [9E9, 9E9, 9E9, 9E9, 9E9, 9E9]];
	VAR jointtarget SDP_259 := [[7.04, 38.15, 2.2, 0, 49.65, -172.96], [9E9, 9E9, 9E9, 9E9, 9E9, 9E9]];
	VAR jointtarget SDP_260 := [[7.05, 37.77, 2.85, 0, 49.38, -177.45], [9E9, 9E9, 9E9, 9E9, 9E9, 9E9]];
	VAR jointtarget SDP_261 := [[7.02, 37.4, 3.5, 0, 49.11, -186.48], [9E9, 9E9, 9E9, 9E9, 9E9, 9E9]];
	VAR jointtarget SDP_262 := [[6.93, 37.04, 4.12, 0, 48.84, -195.57], [9E9, 9E9, 9E9, 9E9, 9E9, 9E9]];
	VAR jointtarget SDP_263 := [[6.78, 36.7, 4.7, 0, 48.6, -204.72], [9E9, 9E9, 9E9, 9E9, 9E9, 9E9]];
	VAR jointtarget SDP_264 := [[6.6, 36.39, 5.23, 0, 48.38, -213.9], [9E9, 9E9, 9E9, 9E9, 9E9, 9E9]];
	VAR jointtarget SDP_265 := [[6.36, 36.12, 5.7, 0, 48.18, -223.14], [9E9, 9E9, 9E9, 9E9, 9E9, 9E9]];
	VAR jointtarget SDP_266 := [[6.09, 35.89, 6.09, 0, 48.02, -232.41], [9E9, 9E9, 9E9, 9E9, 9E9, 9E9]];
	VAR jointtarget SDP_267 := [[5.79, 35.72, 6.39, 0, 47.89, -241.71], [9E9, 9E9, 9E9, 9E9, 9E9, 9E9]];
	VAR jointtarget SDP_268 := [[5.47, 35.6, 6.6, 0, 47.81, -251.03], [9E9, 9E9, 9E9, 9E9, 9E9, 9E9]];
	VAR jointtarget SDP_269 := [[5.13, 35.53, 6.7, 0, 47.76, -260.37], [9E9, 9E9, 9E9, 9E9, 9E9, 9E9]];
	VAR jointtarget SDP_270 := [[4.05, 35.44, 6.86, 0, 47.7, -265.95], [9E9, 9E9, 9E9, 9E9, 9E9, 9E9]];
	VAR jointtarget SDP_271 := [[2.97, 35.37, 6.98, 0, 47.65, -267.03], [9E9, 9E9, 9E9, 9E9, 9E9, 9E9]];
	VAR jointtarget SDP_272 := [[1.89, 35.32, 7.07, 0, 47.61, -268.11], [9E9, 9E9, 9E9, 9E9, 9E9, 9E9]];
	VAR jointtarget SDP_273 := [[0.8, 35.3, 7.11, 0, 47.59, -269.2], [9E9, 9E9, 9E9, 9E9, 9E9, 9E9]];
	VAR jointtarget SDP_274 := [[-0.28, 35.29, 7.12, 0, 47.59, -270.28], [9E9, 9E9, 9E9, 9E9, 9E9, 9E9]];
	VAR jointtarget SDP_275 := [[-1.37, 35.31, 7.09, 0, 47.6, -271.37], [9E9, 9E9, 9E9, 9E9, 9E9, 9E9]];
	VAR jointtarget SDP_276 := [[-2.45, 35.34, 7.03, 0, 47.63, -272.45], [9E9, 9E9, 9E9, 9E9, 9E9, 9E9]];
	VAR jointtarget SDP_277 := [[-3.53, 35.41, 6.92, 0, 47.67, -273.53], [9E9, 9E9, 9E9, 9E9, 9E9, 9E9]];
	VAR jointtarget SDP_278 := [[-4.61, 35.49, 6.78, 0, 47.73, -274.61], [9E9, 9E9, 9E9, 9E9, 9E9, 9E9]];
	VAR jointtarget SDP_279 := [[-5.69, 35.59, 6.61, 0, 47.8, -275.69], [9E9, 9E9, 9E9, 9E9, 9E9, 9E9]];
	VAR jointtarget SDP_280 := [[-5.72, 35.59, 6.6, 0, 47.81, -276.38], [9E9, 9E9, 9E9, 9E9, 9E9, 9E9]];
	VAR jointtarget SDP_281 := [[-5.75, 35.6, 6.59, 0, 47.81, -277.74], [9E9, 9E9, 9E9, 9E9, 9E9, 9E9]];
	VAR jointtarget SDP_282 := [[-5.79, 35.61, 6.58, 0, 47.81, -279.1], [9E9, 9E9, 9E9, 9E9, 9E9, 9E9]];
	VAR jointtarget SDP_283 := [[-5.82, 35.61, 6.57, 0, 47.82, -280.46], [9E9, 9E9, 9E9, 9E9, 9E9, 9E9]];
	VAR jointtarget SDP_284 := [[-5.85, 35.62, 6.56, 0, 47.82, -281.81], [9E9, 9E9, 9E9, 9E9, 9E9, 9E9]];
	VAR jointtarget SDP_285 := [[-5.89, 35.63, 6.54, 0, 47.83, -283.17], [9E9, 9E9, 9E9, 9E9, 9E9, 9E9]];
	VAR jointtarget SDP_286 := [[-5.92, 35.64, 6.53, 0, 47.84, -284.53], [9E9, 9E9, 9E9, 9E9, 9E9, 9E9]];
	VAR jointtarget SDP_287 := [[-5.95, 35.65, 6.51, 0, 47.84, -285.88], [9E9, 9E9, 9E9, 9E9, 9E9, 9E9]];
	VAR jointtarget SDP_288 := [[-5.98, 35.66, 6.49, 0, 47.85, -287.24], [9E9, 9E9, 9E9, 9E9, 9E9, 9E9]];
	VAR jointtarget SDP_289 := [[-6.02, 35.67, 6.47, 0, 47.86, -288.59], [9E9, 9E9, 9E9, 9E9, 9E9, 9E9]];
	VAR jointtarget SDP_290 := [[-6.14, 35.72, 6.39, 0, 47.89, -289.38], [9E9, 9E9, 9E9, 9E9, 9E9, 9E9]];
	VAR jointtarget SDP_291 := [[-6.27, 35.77, 6.31, 0, 47.93, -289.51], [9E9, 9E9, 9E9, 9E9, 9E9, 9E9]];
	VAR jointtarget SDP_292 := [[-6.4, 35.81, 6.22, 0, 47.96, -289.64], [9E9, 9E9, 9E9, 9E9, 9E9, 9E9]];
	VAR jointtarget SDP_293 := [[-6.53, 35.86, 6.14, 0, 48, -289.77], [9E9, 9E9, 9E9, 9E9, 9E9, 9E9]];
	VAR jointtarget SDP_294 := [[-6.66, 35.91, 6.05, 0, 48.03, -289.9], [9E9, 9E9, 9E9, 9E9, 9E9, 9E9]];
	VAR jointtarget SDP_295 := [[-6.78, 35.96, 5.97, 0, 48.07, -290.02], [9E9, 9E9, 9E9, 9E9, 9E9, 9E9]];
	VAR jointtarget SDP_296 := [[-6.91, 36.01, 5.88, 0, 48.11, -290.15], [9E9, 9E9, 9E9, 9E9, 9E9, 9E9]];
	VAR jointtarget SDP_297 := [[-7.04, 36.06, 5.79, 0, 48.14, -290.28], [9E9, 9E9, 9E9, 9E9, 9E9, 9E9]];
	VAR jointtarget SDP_298 := [[-7.16, 36.12, 5.71, 0, 48.18, -290.4], [9E9, 9E9, 9E9, 9E9, 9E9, 9E9]];
	VAR jointtarget SDP_299 := [[-7.29, 36.17, 5.62, 0, 48.22, -290.53], [9E9, 9E9, 9E9, 9E9, 9E9, 9E9]];
	VAR jointtarget SDP_300 := [[-7.55, 36.22, 5.53, 0, 48.25, -280.46], [9E9, 9E9, 9E9, 9E9, 9E9, 9E9]];
	VAR jointtarget SDP_301 := [[-7.8, 36.17, 5.62, 0, 48.22, -260.07], [9E9, 9E9, 9E9, 9E9, 9E9, 9E9]];
	VAR jointtarget SDP_302 := [[-8.03, 36.02, 5.86, 0, 48.11, -239.65], [9E9, 9E9, 9E9, 9E9, 9E9, 9E9]];
	VAR jointtarget SDP_303 := [[-8.2, 35.8, 6.24, 0, 47.96, -219.17], [9E9, 9E9, 9E9, 9E9, 9E9, 9E9]];
	VAR jointtarget SDP_304 := [[-8.28, 35.54, 6.7, 0, 47.76, -198.6], [9E9, 9E9, 9E9, 9E9, 9E9, 9E9]];
	VAR jointtarget SDP_305 := [[-8.27, 35.25, 7.18, 0, 47.56, -177.95], [9E9, 9E9, 9E9, 9E9, 9E9, 9E9]];
	VAR jointtarget SDP_306 := [[-8.17, 34.99, 7.62, 0, 47.38, -157.19], [9E9, 9E9, 9E9, 9E9, 9E9, 9E9]];
	VAR jointtarget SDP_307 := [[-7.98, 34.79, 7.97, 0, 47.24, -136.36], [9E9, 9E9, 9E9, 9E9, 9E9, 9E9]];
	VAR jointtarget SDP_308 := [[-7.74, 34.67, 8.18, 0, 47.15, -115.47], [9E9, 9E9, 9E9, 9E9, 9E9, 9E9]];
	VAR jointtarget SDP_309 := [[-7.47, 34.65, 8.22, 0, 47.14, -94.56], [9E9, 9E9, 9E9, 9E9, 9E9, 9E9]];
	VAR jointtarget SDP_310 := [[-7.34, 34.66, 8.19, 0, 47.15, -84.1], [9E9, 9E9, 9E9, 9E9, 9E9, 9E9]];
	VAR jointtarget SDP_311 := [[-7.2, 34.67, 8.17, 0, 47.16, -83.96], [9E9, 9E9, 9E9, 9E9, 9E9, 9E9]];
	VAR jointtarget SDP_312 := [[-7.06, 34.69, 8.14, 0, 47.17, -83.82], [9E9, 9E9, 9E9, 9E9, 9E9, 9E9]];
	VAR jointtarget SDP_313 := [[-6.92, 34.7, 8.11, 0, 47.18, -83.68], [9E9, 9E9, 9E9, 9E9, 9E9, 9E9]];
	VAR jointtarget SDP_314 := [[-6.79, 34.72, 8.08, 0, 47.2, -83.55], [9E9, 9E9, 9E9, 9E9, 9E9, 9E9]];
	VAR jointtarget SDP_315 := [[-6.65, 34.73, 8.06, 0, 47.21, -83.41], [9E9, 9E9, 9E9, 9E9, 9E9, 9E9]];
	VAR jointtarget SDP_316 := [[-6.51, 34.75, 8.03, 0, 47.22, -83.27], [9E9, 9E9, 9E9, 9E9, 9E9, 9E9]];
	VAR jointtarget SDP_317 := [[-6.38, 34.76, 8, 0, 47.24, -83.14], [9E9, 9E9, 9E9, 9E9, 9E9, 9E9]];
	VAR jointtarget SDP_318 := [[-6.24, 34.78, 7.97, 0, 47.25, -83], [9E9, 9E9, 9E9, 9E9, 9E9, 9E9]];
	VAR jointtarget SDP_319 := [[-6.1, 34.8, 7.94, 0, 47.26, -82.86], [9E9, 9E9, 9E9, 9E9, 9E9, 9E9]];
	VAR jointtarget SDP_320 := [[-6.07, 34.8, 7.93, 0, 47.27, -83.49], [9E9, 9E9, 9E9, 9E9, 9E9, 9E9]];
	VAR jointtarget SDP_321 := [[-6.03, 34.8, 7.92, 0, 47.27, -84.78], [9E9, 9E9, 9E9, 9E9, 9E9, 9E9]];
	VAR jointtarget SDP_322 := [[-6, 34.81, 7.92, 0, 47.27, -86.07], [9E9, 9E9, 9E9, 9E9, 9E9, 9E9]];
	VAR jointtarget SDP_323 := [[-5.97, 34.81, 7.92, 0, 47.27, -87.36], [9E9, 9E9, 9E9, 9E9, 9E9, 9E9]];
	VAR jointtarget SDP_324 := [[-5.93, 34.81, 7.92, 0, 47.27, -88.65], [9E9, 9E9, 9E9, 9E9, 9E9, 9E9]];
	VAR jointtarget SDP_325 := [[-5.9, 34.81, 7.92, 0, 47.27, -89.94], [9E9, 9E9, 9E9, 9E9, 9E9, 9E9]];
	VAR jointtarget SDP_326 := [[-5.86, 34.81, 7.92, 0, 47.27, -91.23], [9E9, 9E9, 9E9, 9E9, 9E9, 9E9]];
	VAR jointtarget SDP_327 := [[-5.83, 34.81, 7.92, 0, 47.27, -92.52], [9E9, 9E9, 9E9, 9E9, 9E9, 9E9]];
	VAR jointtarget SDP_328 := [[-5.79, 34.8, 7.92, 0, 47.27, -93.81], [9E9, 9E9, 9E9, 9E9, 9E9, 9E9]];
	VAR jointtarget SDP_329 := [[-5.76, 34.8, 7.93, 0, 47.27, -95.1], [9E9, 9E9, 9E9, 9E9, 9E9, 9E9]];
	VAR jointtarget SDP_330 := [[-4.6, 34.69, 8.12, 0, 47.19, -94.6], [9E9, 9E9, 9E9, 9E9, 9E9, 9E9]];
	VAR jointtarget SDP_331 := [[-3.43, 34.6, 8.26, 0, 47.13, -93.43], [9E9, 9E9, 9E9, 9E9, 9E9, 9E9]];
	VAR jointtarget SDP_332 := [[-2.26, 34.54, 8.37, 0, 47.09, -92.26], [9E9, 9E9, 9E9, 9E9, 9E9, 9E9]];
	VAR jointtarget SDP_333 := [[-1.09, 34.51, 8.43, 0, 47.06, -91.09], [9E9, 9E9, 9E9, 9E9, 9E9, 9E9]];
	VAR jointtarget SDP_334 := [[0.09, 34.5, 8.45, 0, 47.06, -89.91], [9E9, 9E9, 9E9, 9E9, 9E9, 9E9]];
	VAR jointtarget SDP_335 := [[1.26, 34.51, 8.42, 0, 47.07, -88.74], [9E9, 9E9, 9E9, 9E9, 9E9, 9E9]];
	VAR jointtarget SDP_336 := [[2.43, 34.55, 8.36, 0, 47.09, -87.57], [9E9, 9E9, 9E9, 9E9, 9E9, 9E9]];
	VAR jointtarget SDP_337 := [[3.6, 34.62, 8.25, 0, 47.14, -86.4], [9E9, 9E9, 9E9, 9E9, 9E9, 9E9]];
	VAR jointtarget SDP_338 := [[4.77, 34.7, 8.09, 0, 47.2, -85.23], [9E9, 9E9, 9E9, 9E9, 9E9, 9E9]];
	VAR jointtarget SDP_339 := [[5.93, 34.82, 7.9, 0, 47.28, -84.07], [9E9, 9E9, 9E9, 9E9, 9E9, 9E9]];
	VAR jointtarget SDP_340 := [[6.27, 34.89, 7.78, 0, 47.33, -79.23], [9E9, 9E9, 9E9, 9E9, 9E9, 9E9]];
	VAR jointtarget SDP_341 := [[6.6, 35.01, 7.57, 0, 47.42, -69.9], [9E9, 9E9, 9E9, 9E9, 9E9, 9E9]];
	VAR jointtarget SDP_342 := [[6.9, 35.19, 7.26, 0, 47.54, -60.6], [9E9, 9E9, 9E9, 9E9, 9E9, 9E9]];
	VAR jointtarget SDP_343 := [[7.17, 35.42, 6.87, 0, 47.71, -51.33], [9E9, 9E9, 9E9, 9E9, 9E9, 9E9]];
	VAR jointtarget SDP_344 := [[7.4, 35.69, 6.4, 0, 47.9, -42.1], [9E9, 9E9, 9E9, 9E9, 9E9, 9E9]];
	VAR jointtarget SDP_345 := [[7.59, 36, 5.87, 0, 48.12, -32.91], [9E9, 9E9, 9E9, 9E9, 9E9, 9E9]];
	VAR jointtarget SDP_346 := [[7.73, 36.34, 5.29, 0, 48.37, -23.77], [9E9, 9E9, 9E9, 9E9, 9E9, 9E9]];
	VAR jointtarget SDP_347 := [[7.82, 36.7, 4.67, 0, 48.62, -14.68], [9E9, 9E9, 9E9, 9E9, 9E9, 9E9]];
	VAR jointtarget SDP_348 := [[7.85, 37.07, 4.03, 0, 48.89, -5.65], [9E9, 9E9, 9E9, 9E9, 9E9, 9E9]];
	VAR jointtarget SDP_349 := [[7.83, 37.45, 3.39, 0, 49.17, 3.33], [9E9, 9E9, 9E9, 9E9, 9E9, 9E9]];
	VAR jointtarget SDP_350 := [[7.68, 38.7, 1.22, 0, 50.08, 7.68], [9E9, 9E9, 9E9, 9E9, 9E9, 9E9]];
	VAR jointtarget SDP_351 := [[7.54, 39.97, -1, 0, 51.03, 7.54], [9E9, 9E9, 9E9, 9E9, 9E9, 9E9]];
	VAR jointtarget SDP_352 := [[7.4, 41.25, -3.26, 0, 52, 7.4], [9E9, 9E9, 9E9, 9E9, 9E9, 9E9]];
	VAR jointtarget SDP_353 := [[7.26, 42.56, -5.57, 0, 53.01, 7.26], [9E9, 9E9, 9E9, 9E9, 9E9, 9E9]];
	VAR jointtarget SDP_354 := [[7.13, 43.9, -7.94, 0, 54.04, 7.13], [9E9, 9E9, 9E9, 9E9, 9E9, 9E9]];
	VAR jointtarget SDP_355 := [[7.01, 45.26, -10.37, 0, 55.11, 7.01], [9E9, 9E9, 9E9, 9E9, 9E9, 9E9]];
	VAR jointtarget SDP_356 := [[6.89, 46.65, -12.86, 0, 56.21, 6.89], [9E9, 9E9, 9E9, 9E9, 9E9, 9E9]];
	VAR jointtarget SDP_357 := [[6.77, 48.07, -15.43, 0, 57.36, 6.77], [9E9, 9E9, 9E9, 9E9, 9E9, 9E9]];
	VAR jointtarget SDP_358 := [[6.66, 49.53, -18.08, 0, 58.55, 6.66], [9E9, 9E9, 9E9, 9E9, 9E9, 9E9]];
	VAR jointtarget SDP_359 := [[6.55, 51.04, -20.82, 0, 59.78, 6.55], [9E9, 9E9, 9E9, 9E9, 9E9, 9E9]];
	VAR jointtarget SDP_360 := [[6.55, 51.09, -20.9, 0, 59.82, 5.89], [9E9, 9E9, 9E9, 9E9, 9E9, 9E9]];
	VAR jointtarget SDP_361 := [[6.55, 51.13, -20.98, 0, 59.85, 4.56], [9E9, 9E9, 9E9, 9E9, 9E9, 9E9]];
	VAR jointtarget SDP_362 := [[6.55, 51.18, -21.07, 0, 59.89, 3.24], [9E9, 9E9, 9E9, 9E9, 9E9, 9E9]];
	VAR jointtarget SDP_363 := [[6.54, 51.22, -21.15, 0, 59.93, 1.91], [9E9, 9E9, 9E9, 9E9, 9E9, 9E9]];
	VAR jointtarget SDP_364 := [[6.54, 51.27, -21.23, 0, 59.97, 0.59], [9E9, 9E9, 9E9, 9E9, 9E9, 9E9]];
	VAR jointtarget SDP_365 := [[6.54, 51.31, -21.31, 0, 60, -0.74], [9E9, 9E9, 9E9, 9E9, 9E9, 9E9]];
	VAR jointtarget SDP_366 := [[6.55, 51.36, -21.4, 0, 60.04, -2.06], [9E9, 9E9, 9E9, 9E9, 9E9, 9E9]];
	VAR jointtarget SDP_367 := [[6.55, 51.4, -21.48, 0, 60.08, -3.38], [9E9, 9E9, 9E9, 9E9, 9E9, 9E9]];
	VAR jointtarget SDP_368 := [[6.55, 51.45, -21.56, 0, 60.12, -4.7], [9E9, 9E9, 9E9, 9E9, 9E9, 9E9]];
	VAR jointtarget SDP_369 := [[6.55, 51.49, -21.65, 0, 60.15, -6.03], [9E9, 9E9, 9E9, 9E9, 9E9, 9E9]];
	VAR jointtarget SDP_370 := [[6.57, 51.68, -21.98, 0, 60.3, -6.68], [9E9, 9E9, 9E9, 9E9, 9E9, 9E9]];
	VAR jointtarget SDP_371 := [[6.58, 51.86, -22.32, 0, 60.46, -6.66], [9E9, 9E9, 9E9, 9E9, 9E9, 9E9]];
	VAR jointtarget SDP_372 := [[6.59, 52.04, -22.65, 0, 60.61, -6.65], [9E9, 9E9, 9E9, 9E9, 9E9, 9E9]];
	VAR jointtarget SDP_373 := [[6.6, 52.23, -22.99, 0, 60.76, -6.64], [9E9, 9E9, 9E9, 9E9, 9E9, 9E9]];
	VAR jointtarget SDP_374 := [[6.62, 52.41, -23.33, 0, 60.92, -6.62], [9E9, 9E9, 9E9, 9E9, 9E9, 9E9]];
	VAR jointtarget SDP_375 := [[6.63, 52.6, -23.67, 0, 61.07, -6.61], [9E9, 9E9, 9E9, 9E9, 9E9, 9E9]];
	VAR jointtarget SDP_376 := [[6.64, 52.79, -24.02, 0, 61.23, -6.6], [9E9, 9E9, 9E9, 9E9, 9E9, 9E9]];
	VAR jointtarget SDP_377 := [[6.65, 52.98, -24.36, 0, 61.39, -6.59], [9E9, 9E9, 9E9, 9E9, 9E9, 9E9]];
	VAR jointtarget SDP_378 := [[6.67, 53.17, -24.71, 0, 61.54, -6.57], [9E9, 9E9, 9E9, 9E9, 9E9, 9E9]];
	VAR jointtarget SDP_379 := [[6.68, 53.36, -25.06, 0, 61.7, -6.56], [9E9, 9E9, 9E9, 9E9, 9E9, 9E9]];
	VAR jointtarget SDP_380 := [[6.66, 53.73, -25.74, 0, 62.01, 3.75], [9E9, 9E9, 9E9, 9E9, 9E9, 9E9]];
	VAR jointtarget SDP_381 := [[6.58, 54.07, -26.37, 0, 62.3, 24.31], [9E9, 9E9, 9E9, 9E9, 9E9, 9E9]];
	VAR jointtarget SDP_382 := [[6.43, 54.34, -26.86, 0, 62.52, 44.81], [9E9, 9E9, 9E9, 9E9, 9E9, 9E9]];
	VAR jointtarget SDP_383 := [[6.24, 54.5, -27.16, 0, 62.66, 65.27], [9E9, 9E9, 9E9, 9E9, 9E9, 9E9]];
	VAR jointtarget SDP_384 := [[6.04, 54.53, -27.21, 0, 62.68, 85.71], [9E9, 9E9, 9E9, 9E9, 9E9, 9E9]];
	VAR jointtarget SDP_385 := [[5.84, 54.42, -27.01, 0, 62.59, 106.16], [9E9, 9E9, 9E9, 9E9, 9E9, 9E9]];
	VAR jointtarget SDP_386 := [[5.67, 54.19, -26.59, 0, 62.4, 126.64], [9E9, 9E9, 9E9, 9E9, 9E9, 9E9]];
	VAR jointtarget SDP_387 := [[5.56, 53.87, -26.01, 0, 62.14, 147.18], [9E9, 9E9, 9E9, 9E9, 9E9, 9E9]];
	VAR jointtarget SDP_388 := [[5.52, 53.51, -25.34, 0, 61.83, 167.78], [9E9, 9E9, 9E9, 9E9, 9E9, 9E9]];
	VAR jointtarget SDP_389 := [[5.55, 53.14, -24.66, 0, 61.52, 188.46], [9E9, 9E9, 9E9, 9E9, 9E9, 9E9]];
	VAR jointtarget SDP_390 := [[5.58, 52.96, -24.33, 0, 61.37, 198.82], [9E9, 9E9, 9E9, 9E9, 9E9, 9E9]];
	VAR jointtarget SDP_391 := [[5.62, 52.78, -24.01, 0, 61.22, 198.86], [9E9, 9E9, 9E9, 9E9, 9E9, 9E9]];
	VAR jointtarget SDP_392 := [[5.65, 52.6, -23.68, 0, 61.07, 198.89], [9E9, 9E9, 9E9, 9E9, 9E9, 9E9]];
	VAR jointtarget SDP_393 := [[5.69, 52.43, -23.35, 0, 60.93, 198.93], [9E9, 9E9, 9E9, 9E9, 9E9, 9E9]];
	VAR jointtarget SDP_394 := [[5.72, 52.25, -23.03, 0, 60.78, 198.96], [9E9, 9E9, 9E9, 9E9, 9E9, 9E9]];
	VAR jointtarget SDP_395 := [[5.76, 52.07, -22.71, 0, 60.63, 199], [9E9, 9E9, 9E9, 9E9, 9E9, 9E9]];
	VAR jointtarget SDP_396 := [[5.79, 51.9, -22.39, 0, 60.49, 199.03], [9E9, 9E9, 9E9, 9E9, 9E9, 9E9]];
	VAR jointtarget SDP_397 := [[5.83, 51.72, -22.07, 0, 60.34, 199.07], [9E9, 9E9, 9E9, 9E9, 9E9, 9E9]];
	VAR jointtarget SDP_398 := [[5.87, 51.55, -21.75, 0, 60.2, 199.11], [9E9, 9E9, 9E9, 9E9, 9E9, 9E9]];
	VAR jointtarget SDP_399 := [[5.9, 51.37, -21.43, 0, 60.06, 199.14], [9E9, 9E9, 9E9, 9E9, 9E9, 9E9]];
	VAR jointtarget SDP_400 := [[5.91, 51.33, -21.35, 0, 60.02, 198.49], [9E9, 9E9, 9E9, 9E9, 9E9, 9E9]];
	VAR jointtarget SDP_401 := [[5.92, 51.29, -21.27, 0, 59.98, 197.17], [9E9, 9E9, 9E9, 9E9, 9E9, 9E9]];
	VAR jointtarget SDP_402 := [[5.93, 51.24, -21.19, 0, 59.95, 195.86], [9E9, 9E9, 9E9, 9E9, 9E9, 9E9]];
	VAR jointtarget SDP_403 := [[5.93, 51.2, -21.11, 0, 59.91, 194.54], [9E9, 9E9, 9E9, 9E9, 9E9, 9E9]];
	VAR jointtarget SDP_404 := [[5.94, 51.16, -21.03, 0, 59.88, 193.22], [9E9, 9E9, 9E9, 9E9, 9E9, 9E9]];
	VAR jointtarget SDP_405 := [[5.94, 51.11, -20.95, 0, 59.84, 191.9], [9E9, 9E9, 9E9, 9E9, 9E9, 9E9]];
	VAR jointtarget SDP_406 := [[5.95, 51.07, -20.87, 0, 59.8, 190.58], [9E9, 9E9, 9E9, 9E9, 9E9, 9E9]];
	VAR jointtarget SDP_407 := [[5.95, 51.02, -20.79, 0, 59.77, 189.26], [9E9, 9E9, 9E9, 9E9, 9E9, 9E9]];
	VAR jointtarget SDP_408 := [[5.96, 50.98, -20.71, 0, 59.73, 187.94], [9E9, 9E9, 9E9, 9E9, 9E9, 9E9]];
	VAR jointtarget SDP_409 := [[5.96, 50.93, -20.63, 0, 59.69, 186.62], [9E9, 9E9, 9E9, 9E9, 9E9, 9E9]];
	VAR jointtarget SDP_410 := [[6.05, 49.52, -18.06, 0, 58.54, 186.05], [9E9, 9E9, 9E9, 9E9, 9E9, 9E9]];
	VAR jointtarget SDP_411 := [[6.15, 48.15, -15.57, 0, 57.42, 186.15], [9E9, 9E9, 9E9, 9E9, 9E9, 9E9]];
	VAR jointtarget SDP_412 := [[6.25, 46.81, -13.16, 0, 56.35, 186.25], [9E9, 9E9, 9E9, 9E9, 9E9, 9E9]];
	VAR jointtarget SDP_413 := [[6.35, 45.5, -10.81, 0, 55.31, 186.35], [9E9, 9E9, 9E9, 9E9, 9E9, 9E9]];
	VAR jointtarget SDP_414 := [[6.46, 44.22, -8.52, 0, 54.3, 186.46], [9E9, 9E9, 9E9, 9E9, 9E9, 9E9]];
	VAR jointtarget SDP_415 := [[6.56, 42.97, -6.28, 0, 53.32, 186.56], [9E9, 9E9, 9E9, 9E9, 9E9, 9E9]];
	VAR jointtarget SDP_416 := [[6.68, 41.73, -4.1, 0, 52.37, 186.68], [9E9, 9E9, 9E9, 9E9, 9E9, 9E9]];
	VAR jointtarget SDP_417 := [[6.79, 40.52, -1.96, 0, 51.44, 186.79], [9E9, 9E9, 9E9, 9E9, 9E9, 9E9]];
	VAR jointtarget SDP_418 := [[6.91, 39.32, 0.14, 0, 50.54, 186.91], [9E9, 9E9, 9E9, 9E9, 9E9, 9E9]];
	VAR jointtarget SDP_419 := [[7.04, 38.14, 2.2, 0, 49.67, 187.04], [9E9, 9E9, 9E9, 9E9, 9E9, 9E9]];
	VAR jointtarget SDP_420 := [[7.05, 37.76, 2.85, 0, 49.39, 182.55], [9E9, 9E9, 9E9, 9E9, 9E9, 9E9]];
	VAR jointtarget SDP_421 := [[7.02, 37.39, 3.49, 0, 49.12, 173.52], [9E9, 9E9, 9E9, 9E9, 9E9, 9E9]];
	VAR jointtarget SDP_422 := [[6.93, 37.03, 4.11, 0, 48.86, 164.43], [9E9, 9E9, 9E9, 9E9, 9E9, 9E9]];
	VAR jointtarget SDP_423 := [[6.78, 36.69, 4.7, 0, 48.61, 155.28], [9E9, 9E9, 9E9, 9E9, 9E9, 9E9]];
	VAR jointtarget SDP_424 := [[6.6, 36.38, 5.23, 0, 48.39, 146.1], [9E9, 9E9, 9E9, 9E9, 9E9, 9E9]];
	VAR jointtarget SDP_425 := [[6.36, 36.11, 5.7, 0, 48.2, 136.86], [9E9, 9E9, 9E9, 9E9, 9E9, 9E9]];
	VAR jointtarget SDP_426 := [[6.09, 35.88, 6.08, 0, 48.04, 127.59], [9E9, 9E9, 9E9, 9E9, 9E9, 9E9]];
	VAR jointtarget SDP_427 := [[5.79, 35.7, 6.39, 0, 47.91, 118.29], [9E9, 9E9, 9E9, 9E9, 9E9, 9E9]];
	VAR jointtarget SDP_428 := [[5.47, 35.58, 6.59, 0, 47.82, 108.97], [9E9, 9E9, 9E9, 9E9, 9E9, 9E9]];
	VAR jointtarget SDP_429 := [[5.13, 35.52, 6.7, 0, 47.78, 99.63], [9E9, 9E9, 9E9, 9E9, 9E9, 9E9]];
	VAR jointtarget SDP_430 := [[4.07, 35.43, 6.86, 0, 47.71, 94.07], [9E9, 9E9, 9E9, 9E9, 9E9, 9E9]];
	VAR jointtarget SDP_431 := [[3.01, 35.36, 6.98, 0, 47.66, 93.01], [9E9, 9E9, 9E9, 9E9, 9E9, 9E9]];
	VAR jointtarget SDP_432 := [[1.95, 35.31, 7.06, 0, 47.63, 91.95], [9E9, 9E9, 9E9, 9E9, 9E9, 9E9]];
	VAR jointtarget SDP_433 := [[0.89, 35.28, 7.11, 0, 47.61, 90.89], [9E9, 9E9, 9E9, 9E9, 9E9, 9E9]];
	VAR jointtarget SDP_434 := [[-0.18, 35.28, 7.12, 0, 47.61, 89.82], [9E9, 9E9, 9E9, 9E9, 9E9, 9E9]];
	VAR jointtarget SDP_435 := [[-1.24, 35.29, 7.09, 0, 47.62, 88.76], [9E9, 9E9, 9E9, 9E9, 9E9, 9E9]];
	VAR jointtarget SDP_436 := [[-2.31, 35.33, 7.03, 0, 47.64, 87.69], [9E9, 9E9, 9E9, 9E9, 9E9, 9E9]];
	VAR jointtarget SDP_437 := [[-3.37, 35.38, 6.94, 0, 47.68, 86.63], [9E9, 9E9, 9E9, 9E9, 9E9, 9E9]];
	VAR jointtarget SDP_438 := [[-4.43, 35.46, 6.81, 0, 47.73, 85.57], [9E9, 9E9, 9E9, 9E9, 9E9, 9E9]];
	VAR jointtarget SDP_439 := [[-5.48, 35.56, 6.64, 0, 47.8, 84.52], [9E9, 9E9, 9E9, 9E9, 9E9, 9E9]];
	VAR jointtarget SDP_440 := [[-5.59, 35.56, 6.63, 0, 47.81, 86.6], [9E9, 9E9, 9E9, 9E9, 9E9, 9E9]];
	VAR jointtarget SDP_441 := [[-5.71, 35.56, 6.63, 0, 47.81, 90.88], [9E9, 9E9, 9E9, 9E9, 9E9, 9E9]];
	VAR jointtarget SDP_442 := [[-5.82, 35.55, 6.65, 0, 47.8, 95.15], [9E9, 9E9, 9E9, 9E9, 9E9, 9E9]];
	VAR jointtarget SDP_443 := [[-5.93, 35.53, 6.68, 0, 47.79, 99.43], [9E9, 9E9, 9E9, 9E9, 9E9, 9E9]];
	VAR jointtarget SDP_444 := [[-6.04, 35.5, 6.73, 0, 47.77, 103.71], [9E9, 9E9, 9E9, 9E9, 9E9, 9E9]];
	VAR jointtarget SDP_445 := [[-6.14, 35.47, 6.8, 0, 47.74, 107.99], [9E9, 9E9, 9E9, 9E9, 9E9, 9E9]];
	VAR jointtarget SDP_446 := [[-6.25, 35.42, 6.87, 0, 47.71, 112.27], [9E9, 9E9, 9E9, 9E9, 9E9, 9E9]];
	VAR jointtarget SDP_447 := [[-6.35, 35.37, 6.97, 0, 47.67, 116.56], [9E9, 9E9, 9E9, 9E9, 9E9, 9E9]];
	VAR jointtarget SDP_448 := [[-6.44, 35.3, 7.07, 0, 47.63, 120.85], [9E9, 9E9, 9E9, 9E9, 9E9, 9E9]];
	VAR jointtarget SDP_449 := [[-6.54, 35.24, 7.19, 0, 47.58, 125.15], [9E9, 9E9, 9E9, 9E9, 9E9, 9E9]];
	VAR jointtarget SDP_450 := [[-6.59, 35.19, 7.26, 0, 47.55, 127.29], [9E9, 9E9, 9E9, 9E9, 9E9, 9E9]];
	VAR jointtarget SDP_451 := [[-6.64, 35.15, 7.34, 0, 47.51, 127.23], [9E9, 9E9, 9E9, 9E9, 9E9, 9E9]];
	VAR jointtarget SDP_452 := [[-6.7, 35.1, 7.41, 0, 47.48, 127.18], [9E9, 9E9, 9E9, 9E9, 9E9, 9E9]];
	VAR jointtarget SDP_453 := [[-6.75, 35.06, 7.49, 0, 47.45, 127.12], [9E9, 9E9, 9E9, 9E9, 9E9, 9E9]];
	VAR jointtarget SDP_454 := [[-6.81, 35.02, 7.56, 0, 47.42, 127.07], [9E9, 9E9, 9E9, 9E9, 9E9, 9E9]];
	VAR jointtarget SDP_455 := [[-6.86, 34.97, 7.64, 0, 47.39, 127.01], [9E9, 9E9, 9E9, 9E9, 9E9, 9E9]];
	VAR jointtarget SDP_456 := [[-6.92, 34.93, 7.71, 0, 47.36, 126.96], [9E9, 9E9, 9E9, 9E9, 9E9, 9E9]];
	VAR jointtarget SDP_457 := [[-6.97, 34.89, 7.78, 0, 47.33, 126.91], [9E9, 9E9, 9E9, 9E9, 9E9, 9E9]];
	VAR jointtarget SDP_458 := [[-7.03, 34.84, 7.86, 0, 47.3, 126.85], [9E9, 9E9, 9E9, 9E9, 9E9, 9E9]];
	VAR jointtarget SDP_459 := [[-7.08, 34.8, 7.93, 0, 47.27, 126.8], [9E9, 9E9, 9E9, 9E9, 9E9, 9E9]];
	VAR jointtarget SDP_460 := [[-7.39, 34.66, 8.17, 0, 47.17, 113.1], [9E9, 9E9, 9E9, 9E9, 9E9, 9E9]];
	VAR jointtarget SDP_461 := [[-7.72, 34.69, 8.13, 0, 47.19, 85.99], [9E9, 9E9, 9E9, 9E9, 9E9, 9E9]];
	VAR jointtarget SDP_462 := [[-8.01, 34.87, 7.82, 0, 47.32, 58.93], [9E9, 9E9, 9E9, 9E9, 9E9, 9E9]];
	VAR jointtarget SDP_463 := [[-8.18, 35.16, 7.31, 0, 47.52, 31.98], [9E9, 9E9, 9E9, 9E9, 9E9, 9E9]];
	VAR jointtarget SDP_464 := [[-8.21, 35.51, 6.71, 0, 47.77, 5.18], [9E9, 9E9, 9E9, 9E9, 9E9, 9E9]];
	VAR jointtarget SDP_465 := [[-8.09, 35.84, 6.15, 0, 48.01, -21.48], [9E9, 9E9, 9E9, 9E9, 9E9, 9E9]];
	VAR jointtarget SDP_466 := [[-7.85, 36.08, 5.75, 0, 48.18, -48.01], [9E9, 9E9, 9E9, 9E9, 9E9, 9E9]];
	VAR jointtarget SDP_467 := [[-7.53, 36.17, 5.59, 0, 48.24, -74.47], [9E9, 9E9, 9E9, 9E9, 9E9, 9E9]];
	VAR jointtarget SDP_468 := [[-7.21, 36.1, 5.7, 0, 48.19, -100.93], [9E9, 9E9, 9E9, 9E9, 9E9, 9E9]];
	VAR jointtarget SDP_469 := [[-6.96, 35.89, 6.07, 0, 48.04, -127.44], [9E9, 9E9, 9E9, 9E9, 9E9, 9E9]];
	VAR jointtarget SDP_470 := [[-6.9, 35.82, 6.2, 0, 47.99, -140.78], [9E9, 9E9, 9E9, 9E9, 9E9, 9E9]];
	VAR jointtarget SDP_471 := [[-6.85, 35.74, 6.32, 0, 47.94, -140.72], [9E9, 9E9, 9E9, 9E9, 9E9, 9E9]];
	VAR jointtarget SDP_472 := [[-6.79, 35.67, 6.44, 0, 47.89, -140.67], [9E9, 9E9, 9E9, 9E9, 9E9, 9E9]];
	VAR jointtarget SDP_473 := [[-6.74, 35.6, 6.56, 0, 47.84, -140.62], [9E9, 9E9, 9E9, 9E9, 9E9, 9E9]];
	VAR jointtarget SDP_474 := [[-6.68, 35.53, 6.68, 0, 47.79, -140.56], [9E9, 9E9, 9E9, 9E9, 9E9, 9E9]];
	VAR jointtarget SDP_475 := [[-6.63, 35.46, 6.8, 0, 47.74, -140.51], [9E9, 9E9, 9E9, 9E9, 9E9, 9E9]];
	VAR jointtarget SDP_476 := [[-6.58, 35.39, 6.93, 0, 47.69, -140.45], [9E9, 9E9, 9E9, 9E9, 9E9, 9E9]];
	VAR jointtarget SDP_477 := [[-6.52, 35.32, 7.05, 0, 47.63, -140.4], [9E9, 9E9, 9E9, 9E9, 9E9, 9E9]];
	VAR jointtarget SDP_478 := [[-6.47, 35.25, 7.17, 0, 47.58, -140.34], [9E9, 9E9, 9E9, 9E9, 9E9, 9E9]];
	VAR jointtarget SDP_479 := [[-6.41, 35.18, 7.29, 0, 47.54, -140.29], [9E9, 9E9, 9E9, 9E9, 9E9, 9E9]];
	VAR jointtarget SDP_480 := [[-6.38, 35.15, 7.34, 0, 47.51, -139.16], [9E9, 9E9, 9E9, 9E9, 9E9, 9E9]];
	VAR jointtarget SDP_481 := [[-6.36, 35.12, 7.39, 0, 47.49, -136.92], [9E9, 9E9, 9E9, 9E9, 9E9, 9E9]];
	VAR jointtarget SDP_482 := [[-6.33, 35.09, 7.44, 0, 47.47, -134.69], [9E9, 9E9, 9E9, 9E9, 9E9, 9E9]];
	VAR jointtarget SDP_483 := [[-6.3, 35.06, 7.49, 0, 47.45, -132.45], [9E9, 9E9, 9E9, 9E9, 9E9, 9E9]];
	VAR jointtarget SDP_484 := [[-6.27, 35.03, 7.54, 0, 47.43, -130.22], [9E9, 9E9, 9E9, 9E9, 9E9, 9E9]];
	VAR jointtarget SDP_485 := [[-6.24, 35, 7.58, 0, 47.42, -127.98], [9E9, 9E9, 9E9, 9E9, 9E9, 9E9]];
	VAR jointtarget SDP_486 := [[-6.21, 34.98, 7.62, 0, 47.4, -125.74], [9E9, 9E9, 9E9, 9E9, 9E9, 9E9]];
	VAR jointtarget SDP_487 := [[-6.18, 34.95, 7.66, 0, 47.39, -123.5], [9E9, 9E9, 9E9, 9E9, 9E9, 9E9]];
	VAR jointtarget SDP_488 := [[-6.14, 34.93, 7.7, 0, 47.37, -121.26], [9E9, 9E9, 9E9, 9E9, 9E9, 9E9]];
	VAR jointtarget SDP_489 := [[-6.11, 34.91, 7.73, 0, 47.36, -119.01], [9E9, 9E9, 9E9, 9E9, 9E9, 9E9]];
	VAR jointtarget SDP_490 := [[-6.09, 34.9, 7.75, 0, 47.35, -117.89], [9E9, 9E9, 9E9, 9E9, 9E9, 9E9]];
	VAR jointtarget SDP_491 := [[-6.07, 34.89, 7.76, 0, 47.35, -117.87], [9E9, 9E9, 9E9, 9E9, 9E9, 9E9]];
	VAR jointtarget SDP_492 := [[-6.05, 34.88, 7.78, 0, 47.34, -117.86], [9E9, 9E9, 9E9, 9E9, 9E9, 9E9]];
	VAR jointtarget SDP_493 := [[-6.04, 34.87, 7.8, 0, 47.33, -117.84], [9E9, 9E9, 9E9, 9E9, 9E9, 9E9]];
	VAR jointtarget SDP_494 := [[-6.02, 34.86, 7.81, 0, 47.33, -117.82], [9E9, 9E9, 9E9, 9E9, 9E9, 9E9]];
	VAR jointtarget SDP_495 := [[-6, 34.85, 7.83, 0, 47.32, -117.8], [9E9, 9E9, 9E9, 9E9, 9E9, 9E9]];
	VAR jointtarget SDP_496 := [[-5.98, 34.84, 7.85, 0, 47.32, -117.79], [9E9, 9E9, 9E9, 9E9, 9E9, 9E9]];
	VAR jointtarget SDP_497 := [[-5.97, 34.83, 7.86, 0, 47.31, -117.77], [9E9, 9E9, 9E9, 9E9, 9E9, 9E9]];
	VAR jointtarget SDP_498 := [[-5.95, 34.82, 7.88, 0, 47.3, -117.75], [9E9, 9E9, 9E9, 9E9, 9E9, 9E9]];
	VAR jointtarget SDP_499 := [[-5.93, 34.81, 7.9, 0, 47.3, -117.73], [9E9, 9E9, 9E9, 9E9, 9E9, 9E9]];
	VAR jointtarget SDP_500 := [[-4.75, 34.69, 8.09, 0, 47.22, -94.75], [9E9, 9E9, 9E9, 9E9, 9E9, 9E9]];
	VAR jointtarget SDP_501 := [[-3.57, 34.6, 8.25, 0, 47.15, -93.57], [9E9, 9E9, 9E9, 9E9, 9E9, 9E9]];
	VAR jointtarget SDP_502 := [[-2.38, 34.53, 8.36, 0, 47.11, -92.38], [9E9, 9E9, 9E9, 9E9, 9E9, 9E9]];
	VAR jointtarget SDP_503 := [[-1.19, 34.5, 8.42, 0, 47.08, -91.19], [9E9, 9E9, 9E9, 9E9, 9E9, 9E9]];
	VAR jointtarget SDP_504 := [[0, 34.48, 8.44, 0, 47.07, -90], [9E9, 9E9, 9E9, 9E9, 9E9, 9E9]];
	VAR jointtarget SDP_505 := [[1.19, 34.5, 8.42, 0, 47.08, -88.81], [9E9, 9E9, 9E9, 9E9, 9E9, 9E9]];
	VAR jointtarget SDP_506 := [[2.38, 34.53, 8.36, 0, 47.11, -87.62], [9E9, 9E9, 9E9, 9E9, 9E9, 9E9]];
	VAR jointtarget SDP_507 := [[3.57, 34.6, 8.25, 0, 47.15, -86.43], [9E9, 9E9, 9E9, 9E9, 9E9, 9E9]];
	VAR jointtarget SDP_508 := [[4.75, 34.69, 8.09, 0, 47.22, -85.25], [9E9, 9E9, 9E9, 9E9, 9E9, 9E9]];
	VAR jointtarget SDP_509 := [[5.93, 34.81, 7.9, 0, 47.3, -84.07], [9E9, 9E9, 9E9, 9E9, 9E9, 9E9]];
	VAR jointtarget SDP_510 := [[6.27, 34.87, 7.78, 0, 47.35, -79.23], [9E9, 9E9, 9E9, 9E9, 9E9, 9E9]];
	VAR jointtarget SDP_511 := [[6.6, 35, 7.57, 0, 47.43, -69.9], [9E9, 9E9, 9E9, 9E9, 9E9, 9E9]];
	VAR jointtarget SDP_512 := [[6.9, 35.18, 7.26, 0, 47.56, -60.6], [9E9, 9E9, 9E9, 9E9, 9E9, 9E9]];
	VAR jointtarget SDP_513 := [[7.17, 35.41, 6.87, 0, 47.72, -51.33], [9E9, 9E9, 9E9, 9E9, 9E9, 9E9]];
	VAR jointtarget SDP_514 := [[7.4, 35.68, 6.4, 0, 47.92, -42.1], [9E9, 9E9, 9E9, 9E9, 9E9, 9E9]];
	VAR jointtarget SDP_515 := [[7.59, 35.99, 5.87, 0, 48.14, -32.91], [9E9, 9E9, 9E9, 9E9, 9E9, 9E9]];
	VAR jointtarget SDP_516 := [[7.73, 36.33, 5.29, 0, 48.38, -23.77], [9E9, 9E9, 9E9, 9E9, 9E9, 9E9]];
	VAR jointtarget SDP_517 := [[7.82, 36.69, 4.67, 0, 48.64, -14.68], [9E9, 9E9, 9E9, 9E9, 9E9, 9E9]];
	VAR jointtarget SDP_518 := [[7.85, 37.06, 4.03, 0, 48.91, -5.65], [9E9, 9E9, 9E9, 9E9, 9E9, 9E9]];
	VAR jointtarget SDP_519 := [[7.83, 37.43, 3.39, 0, 49.18, 3.33], [9E9, 9E9, 9E9, 9E9, 9E9, 9E9]];
	VAR jointtarget SDP_520 := [[7.68, 38.66, 1.25, 0, 50.08, 7.68], [9E9, 9E9, 9E9, 9E9, 9E9, 9E9]];
	VAR jointtarget SDP_521 := [[7.54, 39.91, -0.92, 0, 51.01, 7.54], [9E9, 9E9, 9E9, 9E9, 9E9, 9E9]];
	VAR jointtarget SDP_522 := [[7.4, 41.17, -3.14, 0, 51.97, 7.4], [9E9, 9E9, 9E9, 9E9, 9E9, 9E9]];
	VAR jointtarget SDP_523 := [[7.27, 42.46, -5.41, 0, 52.95, 7.27], [9E9, 9E9, 9E9, 9E9, 9E9, 9E9]];
	VAR jointtarget SDP_524 := [[7.15, 43.77, -7.73, 0, 53.96, 7.15], [9E9, 9E9, 9E9, 9E9, 9E9, 9E9]];
	VAR jointtarget SDP_525 := [[7.02, 45.1, -10.11, 0, 55.01, 7.02], [9E9, 9E9, 9E9, 9E9, 9E9, 9E9]];
	VAR jointtarget SDP_526 := [[6.9, 46.46, -12.55, 0, 56.09, 6.9], [9E9, 9E9, 9E9, 9E9, 9E9, 9E9]];
	VAR jointtarget SDP_527 := [[6.79, 47.86, -15.06, 0, 57.21, 6.79], [9E9, 9E9, 9E9, 9E9, 9E9, 9E9]];
	VAR jointtarget SDP_528 := [[6.68, 49.29, -17.65, 0, 58.36, 6.68], [9E9, 9E9, 9E9, 9E9, 9E9, 9E9]];
	VAR jointtarget SDP_529 := [[6.57, 50.76, -20.33, 0, 59.57, 6.57], [9E9, 9E9, 9E9, 9E9, 9E9, 9E9]];
	VAR jointtarget SDP_530 := [[6.56, 50.9, -20.59, 0, 59.69, 8.75], [9E9, 9E9, 9E9, 9E9, 9E9, 9E9]];
	VAR jointtarget SDP_531 := [[6.54, 51.05, -20.86, 0, 59.81, 13.12], [9E9, 9E9, 9E9, 9E9, 9E9, 9E9]];
	VAR jointtarget SDP_532 := [[6.51, 51.19, -21.12, 0, 59.93, 17.48], [9E9, 9E9, 9E9, 9E9, 9E9, 9E9]];
	VAR jointtarget SDP_533 := [[6.48, 51.33, -21.38, 0, 60.04, 21.83], [9E9, 9E9, 9E9, 9E9, 9E9, 9E9]];
	VAR jointtarget SDP_534 := [[6.44, 51.47, -21.62, 0, 60.15, 26.18], [9E9, 9E9, 9E9, 9E9, 9E9, 9E9]];
	VAR jointtarget SDP_535 := [[6.39, 51.6, -21.86, 0, 60.26, 30.52], [9E9, 9E9, 9E9, 9E9, 9E9, 9E9]];
	VAR jointtarget SDP_536 := [[6.34, 51.72, -22.09, 0, 60.36, 34.86], [9E9, 9E9, 9E9, 9E9, 9E9, 9E9]];
	VAR jointtarget SDP_537 := [[6.28, 51.84, -22.3, 0, 60.46, 39.19], [9E9, 9E9, 9E9, 9E9, 9E9, 9E9]];
	VAR jointtarget SDP_538 := [[6.22, 51.95, -22.5, 0, 60.55, 43.51], [9E9, 9E9, 9E9, 9E9, 9E9, 9E9]];
	VAR jointtarget SDP_539 := [[6.15, 52.05, -22.69, 0, 60.64, 47.83], [9E9, 9E9, 9E9, 9E9, 9E9, 9E9]];
	VAR jointtarget SDP_540 := [[6.11, 52.11, -22.8, 0, 60.69, 49.99], [9E9, 9E9, 9E9, 9E9, 9E9, 9E9]];
	VAR jointtarget SDP_541 := [[6.07, 52.17, -22.91, 0, 60.74, 49.95], [9E9, 9E9, 9E9, 9E9, 9E9, 9E9]];
	VAR jointtarget SDP_542 := [[6.03, 52.23, -23.02, 0, 60.79, 49.9], [9E9, 9E9, 9E9, 9E9, 9E9, 9E9]];
	VAR jointtarget SDP_543 := [[5.99, 52.29, -23.13, 0, 60.84, 49.86], [9E9, 9E9, 9E9, 9E9, 9E9, 9E9]];
	VAR jointtarget SDP_544 := [[5.94, 52.35, -23.24, 0, 60.89, 49.82], [9E9, 9E9, 9E9, 9E9, 9E9, 9E9]];
	VAR jointtarget SDP_545 := [[5.9, 52.41, -23.35, 0, 60.94, 49.78], [9E9, 9E9, 9E9, 9E9, 9E9, 9E9]];
	VAR jointtarget SDP_546 := [[5.86, 52.47, -23.46, 0, 60.99, 49.74], [9E9, 9E9, 9E9, 9E9, 9E9, 9E9]];
	VAR jointtarget SDP_547 := [[5.82, 52.53, -23.57, 0, 61.04, 49.7], [9E9, 9E9, 9E9, 9E9, 9E9, 9E9]];
	VAR jointtarget SDP_548 := [[5.78, 52.59, -23.68, 0, 61.09, 49.66], [9E9, 9E9, 9E9, 9E9, 9E9, 9E9]];
	VAR jointtarget SDP_549 := [[5.74, 52.65, -23.79, 0, 61.14, 49.61], [9E9, 9E9, 9E9, 9E9, 9E9, 9E9]];
	VAR jointtarget SDP_550 := [[5.58, 53.02, -24.47, 0, 61.44, 36.07], [9E9, 9E9, 9E9, 9E9, 9E9, 9E9]];
	VAR jointtarget SDP_551 := [[5.54, 53.48, -25.3, 0, 61.82, 9.25], [9E9, 9E9, 9E9, 9E9, 9E9, 9E9]];
	VAR jointtarget SDP_552 := [[5.62, 53.92, -26.12, 0, 62.2, -17.44], [9E9, 9E9, 9E9, 9E9, 9E9, 9E9]];
	VAR jointtarget SDP_553 := [[5.8, 54.26, -26.74, 0, 62.48, -44.04], [9E9, 9E9, 9E9, 9E9, 9E9, 9E9]];
	VAR jointtarget SDP_554 := [[6.04, 54.42, -27.03, 0, 62.61, -70.57], [9E9, 9E9, 9E9, 9E9, 9E9, 9E9]];
	VAR jointtarget SDP_555 := [[6.3, 54.36, -26.92, 0, 62.56, -97.09], [9E9, 9E9, 9E9, 9E9, 9E9, 9E9]];
	VAR jointtarget SDP_556 := [[6.51, 54.1, -26.44, 0, 62.34, -123.65], [9E9, 9E9, 9E9, 9E9, 9E9, 9E9]];
	VAR jointtarget SDP_557 := [[6.64, 53.69, -25.69, 0, 62, -150.3], [9E9, 9E9, 9E9, 9E9, 9E9, 9E9]];
	VAR jointtarget SDP_558 := [[6.66, 53.23, -24.84, 0, 61.61, -177.06], [9E9, 9E9, 9E9, 9E9, 9E9, 9E9]];
	VAR jointtarget SDP_559 := [[6.55, 52.81, -24.07, 0, 61.26, -203.94], [9E9, 9E9, 9E9, 9E9, 9E9, 9E9]];
	VAR jointtarget SDP_560 := [[6.52, 52.73, -23.93, 0, 61.2, -217.36], [9E9, 9E9, 9E9, 9E9, 9E9, 9E9]];
	VAR jointtarget SDP_561 := [[6.48, 52.66, -23.8, 0, 61.14, -217.39], [9E9, 9E9, 9E9, 9E9, 9E9, 9E9]];
	VAR jointtarget SDP_562 := [[6.45, 52.58, -23.66, 0, 61.08, -217.42], [9E9, 9E9, 9E9, 9E9, 9E9, 9E9]];
	VAR jointtarget SDP_563 := [[6.42, 52.51, -23.52, 0, 61.02, -217.46], [9E9, 9E9, 9E9, 9E9, 9E9, 9E9]];
	VAR jointtarget SDP_564 := [[6.39, 52.43, -23.39, 0, 60.95, -217.49], [9E9, 9E9, 9E9, 9E9, 9E9, 9E9]];
	VAR jointtarget SDP_565 := [[6.35, 52.36, -23.25, 0, 60.89, -217.52], [9E9, 9E9, 9E9, 9E9, 9E9, 9E9]];
	VAR jointtarget SDP_566 := [[6.32, 52.29, -23.12, 0, 60.83, -217.56], [9E9, 9E9, 9E9, 9E9, 9E9, 9E9]];
	VAR jointtarget SDP_567 := [[6.29, 52.21, -22.98, 0, 60.77, -217.59], [9E9, 9E9, 9E9, 9E9, 9E9, 9E9]];
	VAR jointtarget SDP_568 := [[6.25, 52.14, -22.85, 0, 60.71, -217.62], [9E9, 9E9, 9E9, 9E9, 9E9, 9E9]];
	VAR jointtarget SDP_569 := [[6.22, 52.07, -22.71, 0, 60.65, -217.66], [9E9, 9E9, 9E9, 9E9, 9E9, 9E9]];
	VAR jointtarget SDP_570 := [[6.17, 51.94, -22.49, 0, 60.55, -215.51], [9E9, 9E9, 9E9, 9E9, 9E9, 9E9]];
	VAR jointtarget SDP_571 := [[6.12, 51.81, -22.25, 0, 60.44, -211.17], [9E9, 9E9, 9E9, 9E9, 9E9, 9E9]];
	VAR jointtarget SDP_572 := [[6.08, 51.68, -22, 0, 60.33, -206.83], [9E9, 9E9, 9E9, 9E9, 9E9, 9E9]];
	VAR jointtarget SDP_573 := [[6.05, 51.54, -21.75, 0, 60.21, -202.47], [9E9, 9E9, 9E9, 9E9, 9E9, 9E9]];
	VAR jointtarget SDP_574 := [[6.02, 51.39, -21.48, 0, 60.09, -198.11], [9E9, 9E9, 9E9, 9E9, 9E9, 9E9]];
	VAR jointtarget SDP_575 := [[6, 51.25, -21.22, 0, 59.97, -193.75], [9E9, 9E9, 9E9, 9E9, 9E9, 9E9]];
	VAR jointtarget SDP_576 := [[5.98, 51.1, -20.95, 0, 59.85, -189.38], [9E9, 9E9, 9E9, 9E9, 9E9, 9E9]];
	VAR jointtarget SDP_577 := [[5.97, 50.95, -20.68, 0, 59.73, -185], [9E9, 9E9, 9E9, 9E9, 9E9, 9E9]];
	VAR jointtarget SDP_578 := [[5.97, 50.8, -20.4, 0, 59.6, -180.61], [9E9, 9E9, 9E9, 9E9, 9E9, 9E9]];
	VAR jointtarget SDP_579 := [[5.98, 50.65, -20.13, 0, 59.48, -176.22], [9E9, 9E9, 9E9, 9E9, 9E9, 9E9]];
	VAR jointtarget SDP_580 := [[6.07, 49.27, -17.63, 0, 58.36, -173.93], [9E9, 9E9, 9E9, 9E9, 9E9, 9E9]];
	VAR jointtarget SDP_581 := [[6.16, 47.93, -15.2, 0, 57.27, -173.84], [9E9, 9E9, 9E9, 9E9, 9E9, 9E9]];
	VAR jointtarget SDP_582 := [[6.26, 46.63, -12.84, 0, 56.22, -173.74], [9E9, 9E9, 9E9, 9E9, 9E9, 9E9]];
	VAR jointtarget SDP_583 := [[6.36, 45.35, -10.55, 0, 55.2, -173.64], [9E9, 9E9, 9E9, 9E9, 9E9, 9E9]];
	VAR jointtarget SDP_584 := [[6.47, 44.09, -8.31, 0, 54.22, -173.53], [9E9, 9E9, 9E9, 9E9, 9E9, 9E9]];
	VAR jointtarget SDP_585 := [[6.57, 42.86, -6.12, 0, 53.26, -173.43], [9E9, 9E9, 9E9, 9E9, 9E9, 9E9]];
	VAR jointtarget SDP_586 := [[6.68, 41.65, -3.98, 0, 52.33, -173.32], [9E9, 9E9, 9E9, 9E9, 9E9, 9E9]];
	VAR jointtarget SDP_587 := [[6.8, 40.46, -1.88, 0, 51.42, -173.2], [9E9, 9E9, 9E9, 9E9, 9E9, 9E9]];
	VAR jointtarget SDP_588 := [[6.92, 39.28, 0.17, 0, 50.54, -173.08], [9E9, 9E9, 9E9, 9E9, 9E9, 9E9]];
	VAR jointtarget SDP_589 := [[7.04, 38.12, 2.19, 0, 49.68, -172.96], [9E9, 9E9, 9E9, 9E9, 9E9, 9E9]];
	VAR jointtarget SDP_590 := [[7.05, 37.75, 2.85, 0, 49.41, -177.45], [9E9, 9E9, 9E9, 9E9, 9E9, 9E9]];
	VAR jointtarget SDP_591 := [[7.02, 37.37, 3.49, 0, 49.14, -186.48], [9E9, 9E9, 9E9, 9E9, 9E9, 9E9]];
	VAR jointtarget SDP_592 := [[6.93, 37.01, 4.11, 0, 48.87, -195.57], [9E9, 9E9, 9E9, 9E9, 9E9, 9E9]];
	VAR jointtarget SDP_593 := [[6.78, 36.67, 4.7, 0, 48.63, -204.72], [9E9, 9E9, 9E9, 9E9, 9E9, 9E9]];
	VAR jointtarget SDP_594 := [[6.6, 36.36, 5.23, 0, 48.41, -213.9], [9E9, 9E9, 9E9, 9E9, 9E9, 9E9]];
	VAR jointtarget SDP_595 := [[6.36, 36.09, 5.69, 0, 48.21, -223.14], [9E9, 9E9, 9E9, 9E9, 9E9, 9E9]];
	VAR jointtarget SDP_596 := [[6.09, 35.87, 6.08, 0, 48.05, -232.41], [9E9, 9E9, 9E9, 9E9, 9E9, 9E9]];
	VAR jointtarget SDP_597 := [[5.79, 35.69, 6.38, 0, 47.93, -241.71], [9E9, 9E9, 9E9, 9E9, 9E9, 9E9]];
	VAR jointtarget SDP_598 := [[5.47, 35.57, 6.59, 0, 47.84, -251.03], [9E9, 9E9, 9E9, 9E9, 9E9, 9E9]];
	VAR jointtarget SDP_599 := [[5.13, 35.51, 6.7, 0, 47.79, -260.37], [9E9, 9E9, 9E9, 9E9, 9E9, 9E9]];
	VAR jointtarget SDP_600 := [[4.05, 35.42, 6.86, 0, 47.73, -265.95], [9E9, 9E9, 9E9, 9E9, 9E9, 9E9]];
	VAR jointtarget SDP_601 := [[2.97, 35.34, 6.98, 0, 47.68, -267.03], [9E9, 9E9, 9E9, 9E9, 9E9, 9E9]];
	VAR jointtarget SDP_602 := [[1.89, 35.3, 7.06, 0, 47.64, -268.11], [9E9, 9E9, 9E9, 9E9, 9E9, 9E9]];
	VAR jointtarget SDP_603 := [[0.8, 35.27, 7.11, 0, 47.62, -269.2], [9E9, 9E9, 9E9, 9E9, 9E9, 9E9]];
	VAR jointtarget SDP_604 := [[-0.28, 35.26, 7.12, 0, 47.62, -270.28], [9E9, 9E9, 9E9, 9E9, 9E9, 9E9]];
	VAR jointtarget SDP_605 := [[-1.37, 35.28, 7.09, 0, 47.63, -271.37], [9E9, 9E9, 9E9, 9E9, 9E9, 9E9]];
	VAR jointtarget SDP_606 := [[-2.45, 35.32, 7.02, 0, 47.66, -272.45], [9E9, 9E9, 9E9, 9E9, 9E9, 9E9]];
	VAR jointtarget SDP_607 := [[-3.53, 35.38, 6.92, 0, 47.7, -273.53], [9E9, 9E9, 9E9, 9E9, 9E9, 9E9]];
	VAR jointtarget SDP_608 := [[-4.61, 35.46, 6.78, 0, 47.76, -274.61], [9E9, 9E9, 9E9, 9E9, 9E9, 9E9]];
	VAR jointtarget SDP_609 := [[-5.69, 35.56, 6.6, 0, 47.83, -275.69], [9E9, 9E9, 9E9, 9E9, 9E9, 9E9]];
	VAR jointtarget SDP_610 := [[-5.72, 35.57, 6.59, 0, 47.84, -276.38], [9E9, 9E9, 9E9, 9E9, 9E9, 9E9]];
	VAR jointtarget SDP_611 := [[-5.75, 35.57, 6.59, 0, 47.84, -277.74], [9E9, 9E9, 9E9, 9E9, 9E9, 9E9]];
	VAR jointtarget SDP_612 := [[-5.79, 35.58, 6.58, 0, 47.85, -279.1], [9E9, 9E9, 9E9, 9E9, 9E9, 9E9]];
	VAR jointtarget SDP_613 := [[-5.82, 35.59, 6.56, 0, 47.85, -280.46], [9E9, 9E9, 9E9, 9E9, 9E9, 9E9]];
	VAR jointtarget SDP_614 := [[-5.85, 35.59, 6.55, 0, 47.86, -281.81], [9E9, 9E9, 9E9, 9E9, 9E9, 9E9]];
	VAR jointtarget SDP_615 := [[-5.89, 35.6, 6.54, 0, 47.86, -283.17], [9E9, 9E9, 9E9, 9E9, 9E9, 9E9]];
	VAR jointtarget SDP_616 := [[-5.92, 35.61, 6.52, 0, 47.87, -284.53], [9E9, 9E9, 9E9, 9E9, 9E9, 9E9]];
	VAR jointtarget SDP_617 := [[-5.95, 35.62, 6.51, 0, 47.87, -285.88], [9E9, 9E9, 9E9, 9E9, 9E9, 9E9]];
	VAR jointtarget SDP_618 := [[-5.98, 35.63, 6.49, 0, 47.88, -287.24], [9E9, 9E9, 9E9, 9E9, 9E9, 9E9]];
	VAR jointtarget SDP_619 := [[-6.02, 35.64, 6.47, 0, 47.89, -288.59], [9E9, 9E9, 9E9, 9E9, 9E9, 9E9]];
	VAR jointtarget SDP_620 := [[-6.14, 35.69, 6.38, 0, 47.92, -289.38], [9E9, 9E9, 9E9, 9E9, 9E9, 9E9]];
	VAR jointtarget SDP_621 := [[-6.27, 35.74, 6.3, 0, 47.96, -289.51], [9E9, 9E9, 9E9, 9E9, 9E9, 9E9]];
	VAR jointtarget SDP_622 := [[-6.4, 35.79, 6.22, 0, 47.99, -289.64], [9E9, 9E9, 9E9, 9E9, 9E9, 9E9]];
	VAR jointtarget SDP_623 := [[-6.53, 35.84, 6.13, 0, 48.03, -289.77], [9E9, 9E9, 9E9, 9E9, 9E9, 9E9]];
	VAR jointtarget SDP_624 := [[-6.66, 35.89, 6.05, 0, 48.06, -289.9], [9E9, 9E9, 9E9, 9E9, 9E9, 9E9]];
	VAR jointtarget SDP_625 := [[-6.78, 35.94, 5.96, 0, 48.1, -290.02], [9E9, 9E9, 9E9, 9E9, 9E9, 9E9]];
	VAR jointtarget SDP_626 := [[-6.91, 35.99, 5.88, 0, 48.14, -290.15], [9E9, 9E9, 9E9, 9E9, 9E9, 9E9]];
	VAR jointtarget SDP_627 := [[-7.04, 36.04, 5.79, 0, 48.17, -290.28], [9E9, 9E9, 9E9, 9E9, 9E9, 9E9]];
	VAR jointtarget SDP_628 := [[-7.16, 36.09, 5.7, 0, 48.21, -290.4], [9E9, 9E9, 9E9, 9E9, 9E9, 9E9]];
	VAR jointtarget SDP_629 := [[-7.29, 36.14, 5.61, 0, 48.25, -290.53], [9E9, 9E9, 9E9, 9E9, 9E9, 9E9]];
	VAR jointtarget SDP_630 := [[-7.55, 36.19, 5.53, 0, 48.28, -280.46], [9E9, 9E9, 9E9, 9E9, 9E9, 9E9]];
	VAR jointtarget SDP_631 := [[-7.8, 36.14, 5.61, 0, 48.25, -260.07], [9E9, 9E9, 9E9, 9E9, 9E9, 9E9]];
	VAR jointtarget SDP_632 := [[-8.03, 36, 5.86, 0, 48.14, -239.65], [9E9, 9E9, 9E9, 9E9, 9E9, 9E9]];
	VAR jointtarget SDP_633 := [[-8.2, 35.78, 6.24, 0, 47.99, -219.17], [9E9, 9E9, 9E9, 9E9, 9E9, 9E9]];
	VAR jointtarget SDP_634 := [[-8.28, 35.51, 6.69, 0, 47.8, -198.6], [9E9, 9E9, 9E9, 9E9, 9E9, 9E9]];
	VAR jointtarget SDP_635 := [[-8.27, 35.23, 7.18, 0, 47.6, -177.95], [9E9, 9E9, 9E9, 9E9, 9E9, 9E9]];
	VAR jointtarget SDP_636 := [[-8.17, 34.97, 7.62, 0, 47.41, -157.19], [9E9, 9E9, 9E9, 9E9, 9E9, 9E9]];
	VAR jointtarget SDP_637 := [[-7.98, 34.76, 7.97, 0, 47.27, -136.36], [9E9, 9E9, 9E9, 9E9, 9E9, 9E9]];
	VAR jointtarget SDP_638 := [[-7.74, 34.64, 8.17, 0, 47.18, -115.47], [9E9, 9E9, 9E9, 9E9, 9E9, 9E9]];
	VAR jointtarget SDP_639 := [[-7.47, 34.62, 8.21, 0, 47.17, -94.56], [9E9, 9E9, 9E9, 9E9, 9E9, 9E9]];
	VAR jointtarget SDP_640 := [[-7.34, 34.63, 8.19, 0, 47.18, -84.1], [9E9, 9E9, 9E9, 9E9, 9E9, 9E9]];
	VAR jointtarget SDP_641 := [[-7.2, 34.65, 8.16, 0, 47.19, -83.96], [9E9, 9E9, 9E9, 9E9, 9E9, 9E9]];
	VAR jointtarget SDP_642 := [[-7.06, 34.66, 8.13, 0, 47.2, -83.82], [9E9, 9E9, 9E9, 9E9, 9E9, 9E9]];
	VAR jointtarget SDP_643 := [[-6.92, 34.68, 8.11, 0, 47.22, -83.68], [9E9, 9E9, 9E9, 9E9, 9E9, 9E9]];
	VAR jointtarget SDP_644 := [[-6.79, 34.69, 8.08, 0, 47.23, -83.55], [9E9, 9E9, 9E9, 9E9, 9E9, 9E9]];
	VAR jointtarget SDP_645 := [[-6.65, 34.71, 8.05, 0, 47.24, -83.41], [9E9, 9E9, 9E9, 9E9, 9E9, 9E9]];
	VAR jointtarget SDP_646 := [[-6.51, 34.72, 8.02, 0, 47.26, -83.27], [9E9, 9E9, 9E9, 9E9, 9E9, 9E9]];
	VAR jointtarget SDP_647 := [[-6.38, 34.74, 7.99, 0, 47.27, -83.14], [9E9, 9E9, 9E9, 9E9, 9E9, 9E9]];
	VAR jointtarget SDP_648 := [[-6.24, 34.75, 7.96, 0, 47.28, -83], [9E9, 9E9, 9E9, 9E9, 9E9, 9E9]];
	VAR jointtarget SDP_649 := [[-6.1, 34.77, 7.93, 0, 47.3, -82.86], [9E9, 9E9, 9E9, 9E9, 9E9, 9E9]];
	VAR jointtarget SDP_650 := [[-6.07, 34.77, 7.93, 0, 47.3, -83.49], [9E9, 9E9, 9E9, 9E9, 9E9, 9E9]];
	VAR jointtarget SDP_651 := [[-6.03, 34.78, 7.92, 0, 47.3, -84.78], [9E9, 9E9, 9E9, 9E9, 9E9, 9E9]];
	VAR jointtarget SDP_652 := [[-6, 34.78, 7.92, 0, 47.3, -86.07], [9E9, 9E9, 9E9, 9E9, 9E9, 9E9]];
	VAR jointtarget SDP_653 := [[-5.97, 34.78, 7.91, 0, 47.31, -87.36], [9E9, 9E9, 9E9, 9E9, 9E9, 9E9]];
	VAR jointtarget SDP_654 := [[-5.93, 34.78, 7.91, 0, 47.31, -88.65], [9E9, 9E9, 9E9, 9E9, 9E9, 9E9]];
	VAR jointtarget SDP_655 := [[-5.9, 34.78, 7.91, 0, 47.31, -89.94], [9E9, 9E9, 9E9, 9E9, 9E9, 9E9]];
	VAR jointtarget SDP_656 := [[-5.86, 34.78, 7.91, 0, 47.31, -91.23], [9E9, 9E9, 9E9, 9E9, 9E9, 9E9]];
	VAR jointtarget SDP_657 := [[-5.83, 34.78, 7.92, 0, 47.3, -92.52], [9E9, 9E9, 9E9, 9E9, 9E9, 9E9]];
	VAR jointtarget SDP_658 := [[-5.79, 34.78, 7.92, 0, 47.3, -93.81], [9E9, 9E9, 9E9, 9E9, 9E9, 9E9]];
	VAR jointtarget SDP_659 := [[-5.76, 34.77, 7.93, 0, 47.3, -95.1], [9E9, 9E9, 9E9, 9E9, 9E9, 9E9]];
	VAR jointtarget SDP_660 := [[-4.6, 34.66, 8.11, 0, 47.22, -94.6], [9E9, 9E9, 9E9, 9E9, 9E9, 9E9]];
	VAR jointtarget SDP_661 := [[-3.43, 34.58, 8.26, 0, 47.16, -93.43], [9E9, 9E9, 9E9, 9E9, 9E9, 9E9]];
	VAR jointtarget SDP_662 := [[-2.26, 34.52, 8.36, 0, 47.12, -92.26], [9E9, 9E9, 9E9, 9E9, 9E9, 9E9]];
	VAR jointtarget SDP_663 := [[-1.09, 34.48, 8.42, 0, 47.1, -91.09], [9E9, 9E9, 9E9, 9E9, 9E9, 9E9]];
	VAR jointtarget SDP_664 := [[0.09, 34.47, 8.44, 0, 47.09, -89.91], [9E9, 9E9, 9E9, 9E9, 9E9, 9E9]];
	VAR jointtarget SDP_665 := [[1.26, 34.48, 8.42, 0, 47.1, -88.74], [9E9, 9E9, 9E9, 9E9, 9E9, 9E9]];
	VAR jointtarget SDP_666 := [[2.43, 34.52, 8.35, 0, 47.13, -87.57], [9E9, 9E9, 9E9, 9E9, 9E9, 9E9]];
	VAR jointtarget SDP_667 := [[3.6, 34.59, 8.24, 0, 47.17, -86.4], [9E9, 9E9, 9E9, 9E9, 9E9, 9E9]];
	VAR jointtarget SDP_668 := [[4.77, 34.68, 8.09, 0, 47.23, -85.23], [9E9, 9E9, 9E9, 9E9, 9E9, 9E9]];
	VAR jointtarget SDP_669 := [[5.93, 34.79, 7.89, 0, 47.31, -84.07], [9E9, 9E9, 9E9, 9E9, 9E9, 9E9]];
	VAR jointtarget SDP_670 := [[6.27, 34.86, 7.78, 0, 47.36, -79.23], [9E9, 9E9, 9E9, 9E9, 9E9, 9E9]];
	VAR jointtarget SDP_671 := [[6.6, 34.98, 7.57, 0, 47.45, -69.9], [9E9, 9E9, 9E9, 9E9, 9E9, 9E9]];
	VAR jointtarget SDP_672 := [[6.9, 35.16, 7.26, 0, 47.58, -60.6], [9E9, 9E9, 9E9, 9E9, 9E9, 9E9]];
	VAR jointtarget SDP_673 := [[7.17, 35.39, 6.87, 0, 47.74, -51.33], [9E9, 9E9, 9E9, 9E9, 9E9, 9E9]];
	VAR jointtarget SDP_674 := [[7.4, 35.67, 6.4, 0, 47.93, -42.1], [9E9, 9E9, 9E9, 9E9, 9E9, 9E9]];
	VAR jointtarget SDP_675 := [[7.59, 35.98, 5.87, 0, 48.15, -32.91], [9E9, 9E9, 9E9, 9E9, 9E9, 9E9]];
	VAR jointtarget SDP_676 := [[7.73, 36.32, 5.29, 0, 48.4, -23.77], [9E9, 9E9, 9E9, 9E9, 9E9, 9E9]];
	VAR jointtarget SDP_677 := [[7.82, 36.68, 4.67, 0, 48.66, -14.68], [9E9, 9E9, 9E9, 9E9, 9E9, 9E9]];
	VAR jointtarget SDP_678 := [[7.85, 37.05, 4.03, 0, 48.92, -5.65], [9E9, 9E9, 9E9, 9E9, 9E9, 9E9]];
	VAR jointtarget SDP_679 := [[7.83, 37.42, 3.38, 0, 49.2, 3.33], [9E9, 9E9, 9E9, 9E9, 9E9, 9E9]];
	VAR jointtarget SDP_680 := [[7.68, 38.67, 1.21, 0, 50.11, 7.68], [9E9, 9E9, 9E9, 9E9, 9E9, 9E9]];
	VAR jointtarget SDP_681 := [[7.54, 39.94, -1, 0, 51.06, 7.54], [9E9, 9E9, 9E9, 9E9, 9E9, 9E9]];
	VAR jointtarget SDP_682 := [[7.4, 41.23, -3.26, 0, 52.03, 7.4], [9E9, 9E9, 9E9, 9E9, 9E9, 9E9]];
	VAR jointtarget SDP_683 := [[7.26, 42.54, -5.58, 0, 53.04, 7.26], [9E9, 9E9, 9E9, 9E9, 9E9, 9E9]];
	VAR jointtarget SDP_684 := [[7.13, 43.87, -7.94, 0, 54.07, 7.13], [9E9, 9E9, 9E9, 9E9, 9E9, 9E9]];
	VAR jointtarget SDP_685 := [[7.01, 45.23, -10.37, 0, 55.14, 7.01], [9E9, 9E9, 9E9, 9E9, 9E9, 9E9]];
	VAR jointtarget SDP_686 := [[6.89, 46.63, -12.87, 0, 56.24, 6.89], [9E9, 9E9, 9E9, 9E9, 9E9, 9E9]];
	VAR jointtarget SDP_687 := [[6.77, 48.05, -15.43, 0, 57.38, 6.77], [9E9, 9E9, 9E9, 9E9, 9E9, 9E9]];
	VAR jointtarget SDP_688 := [[6.66, 49.51, -18.08, 0, 58.57, 6.66], [9E9, 9E9, 9E9, 9E9, 9E9, 9E9]];
	VAR jointtarget SDP_689 := [[6.55, 51.02, -20.83, 0, 59.81, 6.55], [9E9, 9E9, 9E9, 9E9, 9E9, 9E9]];
	VAR jointtarget SDP_690 := [[6.55, 51.06, -20.91, 0, 59.84, 5.89], [9E9, 9E9, 9E9, 9E9, 9E9, 9E9]];
	VAR jointtarget SDP_691 := [[6.55, 51.11, -20.99, 0, 59.88, 4.56], [9E9, 9E9, 9E9, 9E9, 9E9, 9E9]];
	VAR jointtarget SDP_692 := [[6.55, 51.15, -21.07, 0, 59.92, 3.24], [9E9, 9E9, 9E9, 9E9, 9E9, 9E9]];
	VAR jointtarget SDP_693 := [[6.54, 51.2, -21.15, 0, 59.95, 1.91], [9E9, 9E9, 9E9, 9E9, 9E9, 9E9]];
	VAR jointtarget SDP_694 := [[6.54, 51.25, -21.24, 0, 59.99, 0.59], [9E9, 9E9, 9E9, 9E9, 9E9, 9E9]];
	VAR jointtarget SDP_695 := [[6.54, 51.29, -21.32, 0, 60.03, -0.74], [9E9, 9E9, 9E9, 9E9, 9E9, 9E9]];
	VAR jointtarget SDP_696 := [[6.55, 51.34, -21.4, 0, 60.07, -2.06], [9E9, 9E9, 9E9, 9E9, 9E9, 9E9]];
	VAR jointtarget SDP_697 := [[6.55, 51.38, -21.49, 0, 60.1, -3.38], [9E9, 9E9, 9E9, 9E9, 9E9, 9E9]];
	VAR jointtarget SDP_698 := [[6.55, 51.43, -21.57, 0, 60.14, -4.7], [9E9, 9E9, 9E9, 9E9, 9E9, 9E9]];
	VAR jointtarget SDP_699 := [[6.55, 51.47, -21.65, 0, 60.18, -6.03], [9E9, 9E9, 9E9, 9E9, 9E9, 9E9]];
	VAR jointtarget SDP_700 := [[6.57, 51.65, -21.99, 0, 60.33, -6.68], [9E9, 9E9, 9E9, 9E9, 9E9, 9E9]];
	VAR jointtarget SDP_701 := [[6.58, 51.84, -22.32, 0, 60.48, -6.66], [9E9, 9E9, 9E9, 9E9, 9E9, 9E9]];
	VAR jointtarget SDP_702 := [[6.59, 52.02, -22.66, 0, 60.63, -6.65], [9E9, 9E9, 9E9, 9E9, 9E9, 9E9]];
	VAR jointtarget SDP_703 := [[6.6, 52.21, -23, 0, 60.79, -6.64], [9E9, 9E9, 9E9, 9E9, 9E9, 9E9]];
	VAR jointtarget SDP_704 := [[6.62, 52.39, -23.34, 0, 60.94, -6.62], [9E9, 9E9, 9E9, 9E9, 9E9, 9E9]];
	VAR jointtarget SDP_705 := [[6.63, 52.58, -23.68, 0, 61.1, -6.61], [9E9, 9E9, 9E9, 9E9, 9E9, 9E9]];
	VAR jointtarget SDP_706 := [[6.64, 52.77, -24.02, 0, 61.25, -6.6], [9E9, 9E9, 9E9, 9E9, 9E9, 9E9]];
	VAR jointtarget SDP_707 := [[6.65, 52.96, -24.37, 0, 61.41, -6.59], [9E9, 9E9, 9E9, 9E9, 9E9, 9E9]];
	VAR jointtarget SDP_708 := [[6.67, 53.15, -24.71, 0, 61.57, -6.57], [9E9, 9E9, 9E9, 9E9, 9E9, 9E9]];
	VAR jointtarget SDP_709 := [[6.68, 53.34, -25.06, 0, 61.73, -6.56], [9E9, 9E9, 9E9, 9E9, 9E9, 9E9]];
	VAR jointtarget SDP_710 := [[6.66, 53.71, -25.75, 0, 62.04, 3.75], [9E9, 9E9, 9E9, 9E9, 9E9, 9E9]];
	VAR jointtarget SDP_711 := [[6.58, 54.05, -26.38, 0, 62.33, 24.31], [9E9, 9E9, 9E9, 9E9, 9E9, 9E9]];
	VAR jointtarget SDP_712 := [[6.43, 54.32, -26.87, 0, 62.55, 44.81], [9E9, 9E9, 9E9, 9E9, 9E9, 9E9]];
	VAR jointtarget SDP_713 := [[6.24, 54.48, -27.16, 0, 62.68, 65.27], [9E9, 9E9, 9E9, 9E9, 9E9, 9E9]];
	VAR jointtarget SDP_714 := [[6.04, 54.51, -27.21, 0, 62.71, 85.71], [9E9, 9E9, 9E9, 9E9, 9E9, 9E9]];
	VAR jointtarget SDP_715 := [[5.84, 54.4, -27.02, 0, 62.62, 106.16], [9E9, 9E9, 9E9, 9E9, 9E9, 9E9]];
	VAR jointtarget SDP_716 := [[5.67, 54.17, -26.6, 0, 62.43, 126.64], [9E9, 9E9, 9E9, 9E9, 9E9, 9E9]];
	VAR jointtarget SDP_717 := [[5.56, 53.85, -26.02, 0, 62.16, 147.18], [9E9, 9E9, 9E9, 9E9, 9E9, 9E9]];
	VAR jointtarget SDP_718 := [[5.52, 53.49, -25.34, 0, 61.85, 167.78], [9E9, 9E9, 9E9, 9E9, 9E9, 9E9]];
	VAR jointtarget SDP_719 := [[5.55, 53.12, -24.67, 0, 61.55, 188.46], [9E9, 9E9, 9E9, 9E9, 9E9, 9E9]];
	VAR jointtarget SDP_720 := [[5.58, 52.94, -24.34, 0, 61.4, 198.82], [9E9, 9E9, 9E9, 9E9, 9E9, 9E9]];
	VAR jointtarget SDP_721 := [[5.62, 52.76, -24.01, 0, 61.25, 198.86], [9E9, 9E9, 9E9, 9E9, 9E9, 9E9]];
	VAR jointtarget SDP_722 := [[5.65, 52.58, -23.68, 0, 61.1, 198.89], [9E9, 9E9, 9E9, 9E9, 9E9, 9E9]];
	VAR jointtarget SDP_723 := [[5.69, 52.41, -23.36, 0, 60.95, 198.93], [9E9, 9E9, 9E9, 9E9, 9E9, 9E9]];
	VAR jointtarget SDP_724 := [[5.72, 52.23, -23.03, 0, 60.81, 198.96], [9E9, 9E9, 9E9, 9E9, 9E9, 9E9]];
	VAR jointtarget SDP_725 := [[5.76, 52.05, -22.71, 0, 60.66, 199], [9E9, 9E9, 9E9, 9E9, 9E9, 9E9]];
	VAR jointtarget SDP_726 := [[5.79, 51.88, -22.39, 0, 60.51, 199.03], [9E9, 9E9, 9E9, 9E9, 9E9, 9E9]];
	VAR jointtarget SDP_727 := [[5.83, 51.7, -22.07, 0, 60.37, 199.07], [9E9, 9E9, 9E9, 9E9, 9E9, 9E9]];
	VAR jointtarget SDP_728 := [[5.87, 51.53, -21.75, 0, 60.22, 199.11], [9E9, 9E9, 9E9, 9E9, 9E9, 9E9]];
	VAR jointtarget SDP_729 := [[5.9, 51.35, -21.44, 0, 60.08, 199.14], [9E9, 9E9, 9E9, 9E9, 9E9, 9E9]];
	VAR jointtarget SDP_730 := [[5.91, 51.31, -21.36, 0, 60.05, 198.49], [9E9, 9E9, 9E9, 9E9, 9E9, 9E9]];
	VAR jointtarget SDP_731 := [[5.92, 51.27, -21.28, 0, 60.01, 197.17], [9E9, 9E9, 9E9, 9E9, 9E9, 9E9]];
	VAR jointtarget SDP_732 := [[5.93, 51.22, -21.2, 0, 59.97, 195.86], [9E9, 9E9, 9E9, 9E9, 9E9, 9E9]];
	VAR jointtarget SDP_733 := [[5.93, 51.18, -21.12, 0, 59.94, 194.54], [9E9, 9E9, 9E9, 9E9, 9E9, 9E9]];
	VAR jointtarget SDP_734 := [[5.94, 51.14, -21.04, 0, 59.9, 193.22], [9E9, 9E9, 9E9, 9E9, 9E9, 9E9]];
	VAR jointtarget SDP_735 := [[5.94, 51.09, -20.96, 0, 59.87, 191.9], [9E9, 9E9, 9E9, 9E9, 9E9, 9E9]];
	VAR jointtarget SDP_736 := [[5.95, 51.05, -20.88, 0, 59.83, 190.58], [9E9, 9E9, 9E9, 9E9, 9E9, 9E9]];
	VAR jointtarget SDP_737 := [[5.95, 51, -20.79, 0, 59.79, 189.26], [9E9, 9E9, 9E9, 9E9, 9E9, 9E9]];
	VAR jointtarget SDP_738 := [[5.96, 50.96, -20.71, 0, 59.76, 187.94], [9E9, 9E9, 9E9, 9E9, 9E9, 9E9]];
	VAR jointtarget SDP_739 := [[5.96, 50.91, -20.63, 0, 59.72, 186.62], [9E9, 9E9, 9E9, 9E9, 9E9, 9E9]];
	VAR jointtarget SDP_740 := [[6.05, 49.5, -18.06, 0, 58.56, 186.05], [9E9, 9E9, 9E9, 9E9, 9E9, 9E9]];
	VAR jointtarget SDP_741 := [[6.15, 48.13, -15.58, 0, 57.45, 186.15], [9E9, 9E9, 9E9, 9E9, 9E9, 9E9]];
	VAR jointtarget SDP_742 := [[6.25, 46.79, -13.16, 0, 56.37, 186.25], [9E9, 9E9, 9E9, 9E9, 9E9, 9E9]];
	VAR jointtarget SDP_743 := [[6.35, 45.48, -10.81, 0, 55.33, 186.35], [9E9, 9E9, 9E9, 9E9, 9E9, 9E9]];
	VAR jointtarget SDP_744 := [[6.46, 44.2, -8.52, 0, 54.32, 186.46], [9E9, 9E9, 9E9, 9E9, 9E9, 9E9]];
	VAR jointtarget SDP_745 := [[6.56, 42.94, -6.29, 0, 53.35, 186.56], [9E9, 9E9, 9E9, 9E9, 9E9, 9E9]];
	VAR jointtarget SDP_746 := [[6.68, 41.71, -4.1, 0, 52.4, 186.68], [9E9, 9E9, 9E9, 9E9, 9E9, 9E9]];
	VAR jointtarget SDP_747 := [[6.79, 40.49, -1.96, 0, 51.47, 186.79], [9E9, 9E9, 9E9, 9E9, 9E9, 9E9]];
	VAR jointtarget SDP_748 := [[6.91, 39.29, 0.13, 0, 50.57, 186.91], [9E9, 9E9, 9E9, 9E9, 9E9, 9E9]];
	VAR jointtarget SDP_749 := [[7.04, 38.11, 2.19, 0, 49.7, 187.04], [9E9, 9E9, 9E9, 9E9, 9E9, 9E9]];
	VAR jointtarget SDP_750 := [[7.05, 37.73, 2.84, 0, 49.42, 182.55], [9E9, 9E9, 9E9, 9E9, 9E9, 9E9]];
	VAR jointtarget SDP_751 := [[7.02, 37.36, 3.49, 0, 49.15, 173.52], [9E9, 9E9, 9E9, 9E9, 9E9, 9E9]];
	VAR jointtarget SDP_752 := [[6.93, 37, 4.11, 0, 48.89, 164.43], [9E9, 9E9, 9E9, 9E9, 9E9, 9E9]];
	VAR jointtarget SDP_753 := [[6.78, 36.66, 4.69, 0, 48.64, 155.28], [9E9, 9E9, 9E9, 9E9, 9E9, 9E9]];
	VAR jointtarget SDP_754 := [[6.6, 36.35, 5.23, 0, 48.42, 146.1], [9E9, 9E9, 9E9, 9E9, 9E9, 9E9]];
	VAR jointtarget SDP_755 := [[6.36, 36.08, 5.69, 0, 48.23, 136.86], [9E9, 9E9, 9E9, 9E9, 9E9, 9E9]];
	VAR jointtarget SDP_756 := [[6.09, 35.85, 6.08, 0, 48.07, 127.59], [9E9, 9E9, 9E9, 9E9, 9E9, 9E9]];
	VAR jointtarget SDP_757 := [[5.79, 35.68, 6.38, 0, 47.94, 118.29], [9E9, 9E9, 9E9, 9E9, 9E9, 9E9]];
	VAR jointtarget SDP_758 := [[5.47, 35.56, 6.59, 0, 47.85, 108.97], [9E9, 9E9, 9E9, 9E9, 9E9, 9E9]];
	VAR jointtarget SDP_759 := [[5.13, 35.49, 6.7, 0, 47.81, 99.63], [9E9, 9E9, 9E9, 9E9, 9E9, 9E9]];
	VAR jointtarget SDP_760 := [[4.07, 35.4, 6.85, 0, 47.75, 94.07], [9E9, 9E9, 9E9, 9E9, 9E9, 9E9]];
	VAR jointtarget SDP_761 := [[3.01, 35.33, 6.97, 0, 47.7, 93.01], [9E9, 9E9, 9E9, 9E9, 9E9, 9E9]];
	VAR jointtarget SDP_762 := [[1.95, 35.28, 7.05, 0, 47.66, 91.95], [9E9, 9E9, 9E9, 9E9, 9E9, 9E9]];
	VAR jointtarget SDP_763 := [[0.89, 35.26, 7.1, 0, 47.64, 90.89], [9E9, 9E9, 9E9, 9E9, 9E9, 9E9]];
	VAR jointtarget SDP_764 := [[-0.18, 35.25, 7.11, 0, 47.64, 89.82], [9E9, 9E9, 9E9, 9E9, 9E9, 9E9]];
	VAR jointtarget SDP_765 := [[-1.24, 35.26, 7.09, 0, 47.65, 88.76], [9E9, 9E9, 9E9, 9E9, 9E9, 9E9]];
	VAR jointtarget SDP_766 := [[-2.31, 35.3, 7.03, 0, 47.67, 87.69], [9E9, 9E9, 9E9, 9E9, 9E9, 9E9]];
	VAR jointtarget SDP_767 := [[-3.37, 35.35, 6.93, 0, 47.71, 86.63], [9E9, 9E9, 9E9, 9E9, 9E9, 9E9]];
	VAR jointtarget SDP_768 := [[-4.43, 35.43, 6.8, 0, 47.77, 85.57], [9E9, 9E9, 9E9, 9E9, 9E9, 9E9]];
	VAR jointtarget SDP_769 := [[-5.48, 35.53, 6.64, 0, 47.84, 84.52], [9E9, 9E9, 9E9, 9E9, 9E9, 9E9]];
	VAR jointtarget SDP_770 := [[-5.59, 35.54, 6.62, 0, 47.84, 86.6], [9E9, 9E9, 9E9, 9E9, 9E9, 9E9]];
	VAR jointtarget SDP_771 := [[-5.71, 35.53, 6.63, 0, 47.84, 90.88], [9E9, 9E9, 9E9, 9E9, 9E9, 9E9]];
	VAR jointtarget SDP_772 := [[-5.82, 35.52, 6.65, 0, 47.83, 95.15], [9E9, 9E9, 9E9, 9E9, 9E9, 9E9]];
	VAR jointtarget SDP_773 := [[-5.93, 35.5, 6.68, 0, 47.82, 99.43], [9E9, 9E9, 9E9, 9E9, 9E9, 9E9]];
	VAR jointtarget SDP_774 := [[-6.04, 35.48, 6.73, 0, 47.8, 103.71], [9E9, 9E9, 9E9, 9E9, 9E9, 9E9]];
	VAR jointtarget SDP_775 := [[-6.14, 35.44, 6.79, 0, 47.77, 107.99], [9E9, 9E9, 9E9, 9E9, 9E9, 9E9]];
	VAR jointtarget SDP_776 := [[-6.25, 35.39, 6.87, 0, 47.74, 112.27], [9E9, 9E9, 9E9, 9E9, 9E9, 9E9]];
	VAR jointtarget SDP_777 := [[-6.35, 35.34, 6.96, 0, 47.7, 116.56], [9E9, 9E9, 9E9, 9E9, 9E9, 9E9]];
	VAR jointtarget SDP_778 := [[-6.44, 35.28, 7.07, 0, 47.66, 120.85], [9E9, 9E9, 9E9, 9E9, 9E9, 9E9]];
	VAR jointtarget SDP_779 := [[-6.54, 35.21, 7.18, 0, 47.61, 125.15], [9E9, 9E9, 9E9, 9E9, 9E9, 9E9]];
	VAR jointtarget SDP_780 := [[-6.59, 35.16, 7.26, 0, 47.58, 127.29], [9E9, 9E9, 9E9, 9E9, 9E9, 9E9]];
	VAR jointtarget SDP_781 := [[-6.64, 35.12, 7.33, 0, 47.55, 127.23], [9E9, 9E9, 9E9, 9E9, 9E9, 9E9]];
	VAR jointtarget SDP_782 := [[-6.7, 35.08, 7.41, 0, 47.51, 127.18], [9E9, 9E9, 9E9, 9E9, 9E9, 9E9]];
	VAR jointtarget SDP_783 := [[-6.75, 35.03, 7.48, 0, 47.48, 127.12], [9E9, 9E9, 9E9, 9E9, 9E9, 9E9]];
	VAR jointtarget SDP_784 := [[-6.81, 34.99, 7.56, 0, 47.45, 127.07], [9E9, 9E9, 9E9, 9E9, 9E9, 9E9]];
	VAR jointtarget SDP_785 := [[-6.86, 34.95, 7.63, 0, 47.42, 127.01], [9E9, 9E9, 9E9, 9E9, 9E9, 9E9]];
	VAR jointtarget SDP_786 := [[-6.92, 34.9, 7.7, 0, 47.39, 126.96], [9E9, 9E9, 9E9, 9E9, 9E9, 9E9]];
	VAR jointtarget SDP_787 := [[-6.97, 34.86, 7.78, 0, 47.36, 126.91], [9E9, 9E9, 9E9, 9E9, 9E9, 9E9]];
	VAR jointtarget SDP_788 := [[-7.03, 34.82, 7.85, 0, 47.33, 126.85], [9E9, 9E9, 9E9, 9E9, 9E9, 9E9]];
	VAR jointtarget SDP_789 := [[-7.08, 34.77, 7.93, 0, 47.3, 126.8], [9E9, 9E9, 9E9, 9E9, 9E9, 9E9]];
	VAR jointtarget SDP_790 := [[-7.39, 34.64, 8.16, 0, 47.2, 113.1], [9E9, 9E9, 9E9, 9E9, 9E9, 9E9]];
	VAR jointtarget SDP_791 := [[-7.72, 34.66, 8.12, 0, 47.22, 85.99], [9E9, 9E9, 9E9, 9E9, 9E9, 9E9]];
	VAR jointtarget SDP_792 := [[-8.01, 34.84, 7.81, 0, 47.35, 58.93], [9E9, 9E9, 9E9, 9E9, 9E9, 9E9]];
	VAR jointtarget SDP_793 := [[-8.18, 35.14, 7.31, 0, 47.56, 31.98], [9E9, 9E9, 9E9, 9E9, 9E9, 9E9]];
	VAR jointtarget SDP_794 := [[-8.21, 35.49, 6.71, 0, 47.8, 5.18], [9E9, 9E9, 9E9, 9E9, 9E9, 9E9]];
	VAR jointtarget SDP_795 := [[-8.09, 35.81, 6.15, 0, 48.04, -21.48], [9E9, 9E9, 9E9, 9E9, 9E9, 9E9]];
	VAR jointtarget SDP_796 := [[-7.85, 36.05, 5.74, 0, 48.21, -48.01], [9E9, 9E9, 9E9, 9E9, 9E9, 9E9]];
	VAR jointtarget SDP_797 := [[-7.53, 36.14, 5.58, 0, 48.27, -74.47], [9E9, 9E9, 9E9, 9E9, 9E9, 9E9]];
	VAR jointtarget SDP_798 := [[-7.21, 36.08, 5.7, 0, 48.22, -100.93], [9E9, 9E9, 9E9, 9E9, 9E9, 9E9]];
	VAR jointtarget SDP_799 := [[-6.96, 35.86, 6.07, 0, 48.07, -127.44], [9E9, 9E9, 9E9, 9E9, 9E9, 9E9]];
	VAR jointtarget SDP_800 := [[-6.9, 35.79, 6.19, 0, 48.02, -140.78], [9E9, 9E9, 9E9, 9E9, 9E9, 9E9]];
	VAR jointtarget SDP_801 := [[-6.85, 35.72, 6.31, 0, 47.97, -140.72], [9E9, 9E9, 9E9, 9E9, 9E9, 9E9]];
	VAR jointtarget SDP_802 := [[-6.79, 35.65, 6.44, 0, 47.92, -140.67], [9E9, 9E9, 9E9, 9E9, 9E9, 9E9]];
	VAR jointtarget SDP_803 := [[-6.74, 35.58, 6.56, 0, 47.87, -140.62], [9E9, 9E9, 9E9, 9E9, 9E9, 9E9]];
	VAR jointtarget SDP_804 := [[-6.68, 35.5, 6.68, 0, 47.82, -140.56], [9E9, 9E9, 9E9, 9E9, 9E9, 9E9]];
	VAR jointtarget SDP_805 := [[-6.63, 35.43, 6.8, 0, 47.77, -140.51], [9E9, 9E9, 9E9, 9E9, 9E9, 9E9]];
	VAR jointtarget SDP_806 := [[-6.58, 35.36, 6.92, 0, 47.72, -140.45], [9E9, 9E9, 9E9, 9E9, 9E9, 9E9]];
	VAR jointtarget SDP_807 := [[-6.52, 35.29, 7.04, 0, 47.67, -140.4], [9E9, 9E9, 9E9, 9E9, 9E9, 9E9]];
	VAR jointtarget SDP_808 := [[-6.47, 35.22, 7.16, 0, 47.62, -140.34], [9E9, 9E9, 9E9, 9E9, 9E9, 9E9]];
	VAR jointtarget SDP_809 := [[-6.41, 35.15, 7.28, 0, 47.57, -140.29], [9E9, 9E9, 9E9, 9E9, 9E9, 9E9]];
	VAR jointtarget SDP_810 := [[-6.38, 35.12, 7.34, 0, 47.54, -139.16], [9E9, 9E9, 9E9, 9E9, 9E9, 9E9]];
	VAR jointtarget SDP_811 := [[-6.36, 35.09, 7.39, 0, 47.52, -136.92], [9E9, 9E9, 9E9, 9E9, 9E9, 9E9]];
	VAR jointtarget SDP_812 := [[-6.33, 35.06, 7.44, 0, 47.5, -134.69], [9E9, 9E9, 9E9, 9E9, 9E9, 9E9]];
	VAR jointtarget SDP_813 := [[-6.3, 35.03, 7.49, 0, 47.48, -132.45], [9E9, 9E9, 9E9, 9E9, 9E9, 9E9]];
	VAR jointtarget SDP_814 := [[-6.27, 35, 7.53, 0, 47.47, -130.22], [9E9, 9E9, 9E9, 9E9, 9E9, 9E9]];
	VAR jointtarget SDP_815 := [[-6.24, 34.98, 7.58, 0, 47.45, -127.98], [9E9, 9E9, 9E9, 9E9, 9E9, 9E9]];
	VAR jointtarget SDP_816 := [[-6.21, 34.95, 7.62, 0, 47.43, -125.74], [9E9, 9E9, 9E9, 9E9, 9E9, 9E9]];
	VAR jointtarget SDP_817 := [[-6.18, 34.93, 7.66, 0, 47.42, -123.5], [9E9, 9E9, 9E9, 9E9, 9E9, 9E9]];
	VAR jointtarget SDP_818 := [[-6.14, 34.9, 7.69, 0, 47.4, -121.26], [9E9, 9E9, 9E9, 9E9, 9E9, 9E9]];
	VAR jointtarget SDP_819 := [[-6.11, 34.88, 7.73, 0, 47.39, -119.01], [9E9, 9E9, 9E9, 9E9, 9E9, 9E9]];
	VAR jointtarget SDP_820 := [[-6.09, 34.87, 7.74, 0, 47.38, -117.89], [9E9, 9E9, 9E9, 9E9, 9E9, 9E9]];
	VAR jointtarget SDP_821 := [[-6.07, 34.86, 7.76, 0, 47.38, -117.87], [9E9, 9E9, 9E9, 9E9, 9E9, 9E9]];
	VAR jointtarget SDP_822 := [[-6.05, 34.85, 7.78, 0, 47.37, -117.86], [9E9, 9E9, 9E9, 9E9, 9E9, 9E9]];
	VAR jointtarget SDP_823 := [[-6.04, 34.84, 7.79, 0, 47.37, -117.84], [9E9, 9E9, 9E9, 9E9, 9E9, 9E9]];
	VAR jointtarget SDP_824 := [[-6.02, 34.83, 7.81, 0, 47.36, -117.82], [9E9, 9E9, 9E9, 9E9, 9E9, 9E9]];
	VAR jointtarget SDP_825 := [[-6, 34.82, 7.83, 0, 47.35, -117.8], [9E9, 9E9, 9E9, 9E9, 9E9, 9E9]];
	VAR jointtarget SDP_826 := [[-5.98, 34.81, 7.84, 0, 47.35, -117.79], [9E9, 9E9, 9E9, 9E9, 9E9, 9E9]];
	VAR jointtarget SDP_827 := [[-5.97, 34.8, 7.86, 0, 47.34, -117.77], [9E9, 9E9, 9E9, 9E9, 9E9, 9E9]];
	VAR jointtarget SDP_828 := [[-5.95, 34.79, 7.87, 0, 47.34, -117.75], [9E9, 9E9, 9E9, 9E9, 9E9, 9E9]];
	VAR jointtarget SDP_829 := [[-5.93, 34.78, 7.89, 0, 47.33, -117.73], [9E9, 9E9, 9E9, 9E9, 9E9, 9E9]];
	VAR jointtarget SDP_830 := [[-4.75, 34.66, 8.09, 0, 47.25, -94.75], [9E9, 9E9, 9E9, 9E9, 9E9, 9E9]];
	VAR jointtarget SDP_831 := [[-3.57, 34.57, 8.24, 0, 47.18, -93.57], [9E9, 9E9, 9E9, 9E9, 9E9, 9E9]];
	VAR jointtarget SDP_832 := [[-2.38, 34.51, 8.35, 0, 47.14, -92.38], [9E9, 9E9, 9E9, 9E9, 9E9, 9E9]];
	VAR jointtarget SDP_833 := [[-1.19, 34.47, 8.42, 0, 47.11, -91.19], [9E9, 9E9, 9E9, 9E9, 9E9, 9E9]];
	VAR jointtarget SDP_834 := [[0, 34.46, 8.44, 0, 47.1, -90], [9E9, 9E9, 9E9, 9E9, 9E9, 9E9]];
	VAR jointtarget SDP_835 := [[1.19, 34.47, 8.42, 0, 47.11, -88.81], [9E9, 9E9, 9E9, 9E9, 9E9, 9E9]];
	VAR jointtarget SDP_836 := [[2.38, 34.51, 8.35, 0, 47.14, -87.62], [9E9, 9E9, 9E9, 9E9, 9E9, 9E9]];
	VAR jointtarget SDP_837 := [[3.57, 34.57, 8.24, 0, 47.18, -86.43], [9E9, 9E9, 9E9, 9E9, 9E9, 9E9]];
	VAR jointtarget SDP_838 := [[4.75, 34.66, 8.09, 0, 47.25, -85.25], [9E9, 9E9, 9E9, 9E9, 9E9, 9E9]];
	VAR jointtarget SDP_839 := [[5.93, 34.78, 7.89, 0, 47.33, -84.07], [9E9, 9E9, 9E9, 9E9, 9E9, 9E9]];
	VAR jointtarget SDP_840 := [[6.27, 34.85, 7.78, 0, 47.38, -79.23], [9E9, 9E9, 9E9, 9E9, 9E9, 9E9]];
	VAR jointtarget SDP_841 := [[6.6, 34.97, 7.56, 0, 47.47, -69.9], [9E9, 9E9, 9E9, 9E9, 9E9, 9E9]];
	VAR jointtarget SDP_842 := [[6.9, 35.15, 7.26, 0, 47.59, -60.6], [9E9, 9E9, 9E9, 9E9, 9E9, 9E9]];
	VAR jointtarget SDP_843 := [[7.17, 35.38, 6.87, 0, 47.75, -51.33], [9E9, 9E9, 9E9, 9E9, 9E9, 9E9]];
	VAR jointtarget SDP_844 := [[7.4, 35.65, 6.4, 0, 47.95, -42.1], [9E9, 9E9, 9E9, 9E9, 9E9, 9E9]];
	VAR jointtarget SDP_845 := [[7.59, 35.96, 5.87, 0, 48.17, -32.91], [9E9, 9E9, 9E9, 9E9, 9E9, 9E9]];
	VAR jointtarget SDP_846 := [[7.73, 36.3, 5.28, 0, 48.41, -23.77], [9E9, 9E9, 9E9, 9E9, 9E9, 9E9]];
	VAR jointtarget SDP_847 := [[7.82, 36.66, 4.67, 0, 48.67, -14.68], [9E9, 9E9, 9E9, 9E9, 9E9, 9E9]];
	VAR jointtarget SDP_848 := [[7.85, 37.03, 4.03, 0, 48.94, -5.65], [9E9, 9E9, 9E9, 9E9, 9E9, 9E9]];
	VAR jointtarget SDP_849 := [[7.83, 37.41, 3.38, 0, 49.21, 3.33], [9E9, 9E9, 9E9, 9E9, 9E9, 9E9]];
	VAR jointtarget SDP_850 := [[7.68, 38.64, 1.25, 0, 50.11, 7.68], [9E9, 9E9, 9E9, 9E9, 9E9, 9E9]];
	VAR jointtarget SDP_851 := [[7.54, 39.88, -0.92, 0, 51.04, 7.54], [9E9, 9E9, 9E9, 9E9, 9E9, 9E9]];
	VAR jointtarget SDP_852 := [[7.4, 41.15, -3.14, 0, 51.99, 7.4], [9E9, 9E9, 9E9, 9E9, 9E9, 9E9]];
	VAR jointtarget SDP_853 := [[7.27, 42.43, -5.41, 0, 52.98, 7.27], [9E9, 9E9, 9E9, 9E9, 9E9, 9E9]];
	VAR jointtarget SDP_854 := [[7.15, 43.74, -7.73, 0, 53.99, 7.15], [9E9, 9E9, 9E9, 9E9, 9E9, 9E9]];
	VAR jointtarget SDP_855 := [[7.02, 45.08, -10.11, 0, 55.04, 7.02], [9E9, 9E9, 9E9, 9E9, 9E9, 9E9]];
	VAR jointtarget SDP_856 := [[6.9, 46.44, -12.55, 0, 56.11, 6.9], [9E9, 9E9, 9E9, 9E9, 9E9, 9E9]];
	VAR jointtarget SDP_857 := [[6.79, 47.83, -15.07, 0, 57.23, 6.79], [9E9, 9E9, 9E9, 9E9, 9E9, 9E9]];
	VAR jointtarget SDP_858 := [[6.68, 49.26, -17.66, 0, 58.39, 6.68], [9E9, 9E9, 9E9, 9E9, 9E9, 9E9]];
	VAR jointtarget SDP_859 := [[6.57, 50.74, -20.33, 0, 59.59, 6.57], [9E9, 9E9, 9E9, 9E9, 9E9, 9E9]];
	VAR jointtarget SDP_860 := [[6.56, 50.88, -20.6, 0, 59.72, 8.75], [9E9, 9E9, 9E9, 9E9, 9E9, 9E9]];
	VAR jointtarget SDP_861 := [[6.54, 51.03, -20.86, 0, 59.84, 13.12], [9E9, 9E9, 9E9, 9E9, 9E9, 9E9]];
	VAR jointtarget SDP_862 := [[6.51, 51.17, -21.13, 0, 59.95, 17.48], [9E9, 9E9, 9E9, 9E9, 9E9, 9E9]];
	VAR jointtarget SDP_863 := [[6.48, 51.31, -21.38, 0, 60.07, 21.83], [9E9, 9E9, 9E9, 9E9, 9E9, 9E9]];
	VAR jointtarget SDP_864 := [[6.44, 51.45, -21.63, 0, 60.18, 26.18], [9E9, 9E9, 9E9, 9E9, 9E9, 9E9]];
	VAR jointtarget SDP_865 := [[6.39, 51.58, -21.86, 0, 60.29, 30.52], [9E9, 9E9, 9E9, 9E9, 9E9, 9E9]];
	VAR jointtarget SDP_866 := [[6.34, 51.7, -22.09, 0, 60.39, 34.86], [9E9, 9E9, 9E9, 9E9, 9E9, 9E9]];
	VAR jointtarget SDP_867 := [[6.28, 51.82, -22.31, 0, 60.49, 39.19], [9E9, 9E9, 9E9, 9E9, 9E9, 9E9]];
	VAR jointtarget SDP_868 := [[6.22, 51.93, -22.51, 0, 60.58, 43.51], [9E9, 9E9, 9E9, 9E9, 9E9, 9E9]];
	VAR jointtarget SDP_869 := [[6.15, 52.03, -22.7, 0, 60.66, 47.83], [9E9, 9E9, 9E9, 9E9, 9E9, 9E9]];
	VAR jointtarget SDP_870 := [[6.11, 52.09, -22.81, 0, 60.71, 49.99], [9E9, 9E9, 9E9, 9E9, 9E9, 9E9]];
	VAR jointtarget SDP_871 := [[6.07, 52.15, -22.91, 0, 60.76, 49.95], [9E9, 9E9, 9E9, 9E9, 9E9, 9E9]];
	VAR jointtarget SDP_872 := [[6.03, 52.21, -23.02, 0, 60.81, 49.9], [9E9, 9E9, 9E9, 9E9, 9E9, 9E9]];
	VAR jointtarget SDP_873 := [[5.99, 52.27, -23.13, 0, 60.86, 49.86], [9E9, 9E9, 9E9, 9E9, 9E9, 9E9]];
	VAR jointtarget SDP_874 := [[5.94, 52.33, -23.24, 0, 60.91, 49.82], [9E9, 9E9, 9E9, 9E9, 9E9, 9E9]];
	VAR jointtarget SDP_875 := [[5.9, 52.39, -23.35, 0, 60.96, 49.78], [9E9, 9E9, 9E9, 9E9, 9E9, 9E9]];
	VAR jointtarget SDP_876 := [[5.86, 52.45, -23.46, 0, 61.01, 49.74], [9E9, 9E9, 9E9, 9E9, 9E9, 9E9]];
	VAR jointtarget SDP_877 := [[5.82, 52.51, -23.57, 0, 61.06, 49.7], [9E9, 9E9, 9E9, 9E9, 9E9, 9E9]];
	VAR jointtarget SDP_878 := [[5.78, 52.57, -23.68, 0, 61.11, 49.66], [9E9, 9E9, 9E9, 9E9, 9E9, 9E9]];
	VAR jointtarget SDP_879 := [[5.74, 52.63, -23.8, 0, 61.16, 49.61], [9E9, 9E9, 9E9, 9E9, 9E9, 9E9]];
	VAR jointtarget SDP_880 := [[5.58, 53, -24.47, 0, 61.47, 36.07], [9E9, 9E9, 9E9, 9E9, 9E9, 9E9]];
	VAR jointtarget SDP_881 := [[5.54, 53.46, -25.31, 0, 61.85, 9.25], [9E9, 9E9, 9E9, 9E9, 9E9, 9E9]];
	VAR jointtarget SDP_882 := [[5.62, 53.9, -26.13, 0, 62.22, -17.44], [9E9, 9E9, 9E9, 9E9, 9E9, 9E9]];
	VAR jointtarget SDP_883 := [[5.8, 54.24, -26.75, 0, 62.51, -44.04], [9E9, 9E9, 9E9, 9E9, 9E9, 9E9]];
	VAR jointtarget SDP_884 := [[6.04, 54.4, -27.03, 0, 62.64, -70.57], [9E9, 9E9, 9E9, 9E9, 9E9, 9E9]];
	VAR jointtarget SDP_885 := [[6.3, 54.34, -26.93, 0, 62.59, -97.09], [9E9, 9E9, 9E9, 9E9, 9E9, 9E9]];
	VAR jointtarget SDP_886 := [[6.51, 54.08, -26.44, 0, 62.37, -123.65], [9E9, 9E9, 9E9, 9E9, 9E9, 9E9]];
	VAR jointtarget SDP_887 := [[6.64, 53.67, -25.69, 0, 62.03, -150.3], [9E9, 9E9, 9E9, 9E9, 9E9, 9E9]];
	VAR jointtarget SDP_888 := [[6.66, 53.2, -24.84, 0, 61.64, -177.06], [9E9, 9E9, 9E9, 9E9, 9E9, 9E9]];
	VAR jointtarget SDP_889 := [[6.55, 52.78, -24.07, 0, 61.29, -203.94], [9E9, 9E9, 9E9, 9E9, 9E9, 9E9]];
	VAR jointtarget SDP_890 := [[6.52, 52.71, -23.94, 0, 61.23, -217.36], [9E9, 9E9, 9E9, 9E9, 9E9, 9E9]];
	VAR jointtarget SDP_891 := [[6.48, 52.64, -23.8, 0, 61.17, -217.39], [9E9, 9E9, 9E9, 9E9, 9E9, 9E9]];
	VAR jointtarget SDP_892 := [[6.45, 52.56, -23.66, 0, 61.1, -217.42], [9E9, 9E9, 9E9, 9E9, 9E9, 9E9]];
	VAR jointtarget SDP_893 := [[6.42, 52.49, -23.53, 0, 61.04, -217.46], [9E9, 9E9, 9E9, 9E9, 9E9, 9E9]];
	VAR jointtarget SDP_894 := [[6.39, 52.41, -23.39, 0, 60.98, -217.49], [9E9, 9E9, 9E9, 9E9, 9E9, 9E9]];
	VAR jointtarget SDP_895 := [[6.35, 52.34, -23.26, 0, 60.92, -217.52], [9E9, 9E9, 9E9, 9E9, 9E9, 9E9]];
	VAR jointtarget SDP_896 := [[6.32, 52.27, -23.12, 0, 60.86, -217.56], [9E9, 9E9, 9E9, 9E9, 9E9, 9E9]];
	VAR jointtarget SDP_897 := [[6.29, 52.19, -22.99, 0, 60.8, -217.59], [9E9, 9E9, 9E9, 9E9, 9E9, 9E9]];
	VAR jointtarget SDP_898 := [[6.25, 52.12, -22.85, 0, 60.74, -217.62], [9E9, 9E9, 9E9, 9E9, 9E9, 9E9]];
	VAR jointtarget SDP_899 := [[6.22, 52.04, -22.72, 0, 60.67, -217.66], [9E9, 9E9, 9E9, 9E9, 9E9, 9E9]];
	VAR jointtarget SDP_900 := [[6.17, 51.92, -22.49, 0, 60.57, -215.51], [9E9, 9E9, 9E9, 9E9, 9E9, 9E9]];
	VAR jointtarget SDP_901 := [[6.12, 51.79, -22.25, 0, 60.46, -211.17], [9E9, 9E9, 9E9, 9E9, 9E9, 9E9]];
	VAR jointtarget SDP_902 := [[6.08, 51.65, -22.01, 0, 60.35, -206.83], [9E9, 9E9, 9E9, 9E9, 9E9, 9E9]];
	VAR jointtarget SDP_903 := [[6.05, 51.51, -21.75, 0, 60.24, -202.47], [9E9, 9E9, 9E9, 9E9, 9E9, 9E9]];
	VAR jointtarget SDP_904 := [[6.02, 51.37, -21.49, 0, 60.12, -198.11], [9E9, 9E9, 9E9, 9E9, 9E9, 9E9]];
	VAR jointtarget SDP_905 := [[6, 51.22, -21.22, 0, 60, -193.75], [9E9, 9E9, 9E9, 9E9, 9E9, 9E9]];
	VAR jointtarget SDP_906 := [[5.98, 51.08, -20.95, 0, 59.87, -189.38], [9E9, 9E9, 9E9, 9E9, 9E9, 9E9]];
	VAR jointtarget SDP_907 := [[5.97, 50.93, -20.68, 0, 59.75, -185], [9E9, 9E9, 9E9, 9E9, 9E9, 9E9]];
	VAR jointtarget SDP_908 := [[5.97, 50.78, -20.41, 0, 59.63, -180.61], [9E9, 9E9, 9E9, 9E9, 9E9, 9E9]];
	VAR jointtarget SDP_909 := [[5.98, 50.63, -20.14, 0, 59.51, -176.22], [9E9, 9E9, 9E9, 9E9, 9E9, 9E9]];
	VAR jointtarget SDP_910 := [[6.07, 49.25, -17.64, 0, 58.38, -173.93], [9E9, 9E9, 9E9, 9E9, 9E9, 9E9]];
	VAR jointtarget SDP_911 := [[6.16, 47.91, -15.21, 0, 57.3, -173.84], [9E9, 9E9, 9E9, 9E9, 9E9, 9E9]];
	VAR jointtarget SDP_912 := [[6.26, 46.6, -12.85, 0, 56.25, -173.74], [9E9, 9E9, 9E9, 9E9, 9E9, 9E9]];
	VAR jointtarget SDP_913 := [[6.36, 45.32, -10.55, 0, 55.23, -173.64], [9E9, 9E9, 9E9, 9E9, 9E9, 9E9]];
	VAR jointtarget SDP_914 := [[6.47, 44.07, -8.31, 0, 54.24, -173.53], [9E9, 9E9, 9E9, 9E9, 9E9, 9E9]];
	VAR jointtarget SDP_915 := [[6.57, 42.84, -6.12, 0, 53.29, -173.43], [9E9, 9E9, 9E9, 9E9, 9E9, 9E9]];
	VAR jointtarget SDP_916 := [[6.68, 41.63, -3.98, 0, 52.36, -173.32], [9E9, 9E9, 9E9, 9E9, 9E9, 9E9]];
	VAR jointtarget SDP_917 := [[6.8, 40.43, -1.89, 0, 51.45, -173.2], [9E9, 9E9, 9E9, 9E9, 9E9, 9E9]];
	VAR jointtarget SDP_918 := [[6.92, 39.26, 0.17, 0, 50.57, -173.08], [9E9, 9E9, 9E9, 9E9, 9E9, 9E9]];
	VAR jointtarget SDP_919 := [[7.04, 38.1, 2.19, 0, 49.71, -172.96], [9E9, 9E9, 9E9, 9E9, 9E9, 9E9]];
	VAR jointtarget SDP_920 := [[7.05, 37.72, 2.84, 0, 49.44, -177.45], [9E9, 9E9, 9E9, 9E9, 9E9, 9E9]];
	VAR jointtarget SDP_921 := [[7.02, 37.35, 3.49, 0, 49.17, -186.48], [9E9, 9E9, 9E9, 9E9, 9E9, 9E9]];
	VAR jointtarget SDP_922 := [[6.93, 36.99, 4.11, 0, 48.91, -195.57], [9E9, 9E9, 9E9, 9E9, 9E9, 9E9]];
	VAR jointtarget SDP_923 := [[6.78, 36.65, 4.69, 0, 48.66, -204.72], [9E9, 9E9, 9E9, 9E9, 9E9, 9E9]];
	VAR jointtarget SDP_924 := [[6.6, 36.34, 5.22, 0, 48.44, -213.9], [9E9, 9E9, 9E9, 9E9, 9E9, 9E9]];
	VAR jointtarget SDP_925 := [[6.36, 36.07, 5.69, 0, 48.24, -223.14], [9E9, 9E9, 9E9, 9E9, 9E9, 9E9]];
	VAR jointtarget SDP_926 := [[6.09, 35.84, 6.08, 0, 48.08, -232.41], [9E9, 9E9, 9E9, 9E9, 9E9, 9E9]];
	VAR jointtarget SDP_927 := [[5.79, 35.66, 6.38, 0, 47.96, -241.71], [9E9, 9E9, 9E9, 9E9, 9E9, 9E9]];
	VAR jointtarget SDP_928 := [[5.47, 35.54, 6.59, 0, 47.87, -251.03], [9E9, 9E9, 9E9, 9E9, 9E9, 9E9]];
	VAR jointtarget SDP_929 := [[5.13, 35.48, 6.69, 0, 47.83, -260.37], [9E9, 9E9, 9E9, 9E9, 9E9, 9E9]];
	VAR jointtarget SDP_930 := [[4.05, 35.39, 6.85, 0, 47.76, -265.95], [9E9, 9E9, 9E9, 9E9, 9E9, 9E9]];
	VAR jointtarget SDP_931 := [[2.97, 35.32, 6.97, 0, 47.71, -267.03], [9E9, 9E9, 9E9, 9E9, 9E9, 9E9]];
	VAR jointtarget SDP_932 := [[1.89, 35.27, 7.06, 0, 47.68, -268.11], [9E9, 9E9, 9E9, 9E9, 9E9, 9E9]];
	VAR jointtarget SDP_933 := [[0.8, 35.24, 7.1, 0, 47.66, -269.2], [9E9, 9E9, 9E9, 9E9, 9E9, 9E9]];
	VAR jointtarget SDP_934 := [[-0.28, 35.24, 7.11, 0, 47.65, -270.28], [9E9, 9E9, 9E9, 9E9, 9E9, 9E9]];
	VAR jointtarget SDP_935 := [[-1.37, 35.25, 7.08, 0, 47.66, -271.37], [9E9, 9E9, 9E9, 9E9, 9E9, 9E9]];
	VAR jointtarget SDP_936 := [[-2.45, 35.29, 7.02, 0, 47.69, -272.45], [9E9, 9E9, 9E9, 9E9, 9E9, 9E9]];
	VAR jointtarget SDP_937 := [[-3.53, 35.35, 6.91, 0, 47.73, -273.53], [9E9, 9E9, 9E9, 9E9, 9E9, 9E9]];
	VAR jointtarget SDP_938 := [[-4.61, 35.43, 6.77, 0, 47.79, -274.61], [9E9, 9E9, 9E9, 9E9, 9E9, 9E9]];
	VAR jointtarget SDP_939 := [[-5.69, 35.54, 6.6, 0, 47.87, -275.69], [9E9, 9E9, 9E9, 9E9, 9E9, 9E9]];
	VAR jointtarget SDP_940 := [[-5.72, 35.54, 6.59, 0, 47.87, -276.38], [9E9, 9E9, 9E9, 9E9, 9E9, 9E9]];
	VAR jointtarget SDP_941 := [[-5.75, 35.55, 6.58, 0, 47.87, -277.74], [9E9, 9E9, 9E9, 9E9, 9E9, 9E9]];
	VAR jointtarget SDP_942 := [[-5.79, 35.55, 6.57, 0, 47.88, -279.1], [9E9, 9E9, 9E9, 9E9, 9E9, 9E9]];
	VAR jointtarget SDP_943 := [[-5.82, 35.56, 6.56, 0, 47.88, -280.46], [9E9, 9E9, 9E9, 9E9, 9E9, 9E9]];
	VAR jointtarget SDP_944 := [[-5.85, 35.57, 6.55, 0, 47.89, -281.81], [9E9, 9E9, 9E9, 9E9, 9E9, 9E9]];
	VAR jointtarget SDP_945 := [[-5.89, 35.57, 6.53, 0, 47.89, -283.17], [9E9, 9E9, 9E9, 9E9, 9E9, 9E9]];
	VAR jointtarget SDP_946 := [[-5.92, 35.58, 6.52, 0, 47.9, -284.53], [9E9, 9E9, 9E9, 9E9, 9E9, 9E9]];
	VAR jointtarget SDP_947 := [[-5.95, 35.59, 6.5, 0, 47.91, -285.88], [9E9, 9E9, 9E9, 9E9, 9E9, 9E9]];
	VAR jointtarget SDP_948 := [[-5.98, 35.6, 6.48, 0, 47.91, -287.24], [9E9, 9E9, 9E9, 9E9, 9E9, 9E9]];
	VAR jointtarget SDP_949 := [[-6.02, 35.62, 6.46, 0, 47.92, -288.59], [9E9, 9E9, 9E9, 9E9, 9E9, 9E9]];
	VAR jointtarget SDP_950 := [[-6.14, 35.66, 6.38, 0, 47.96, -289.38], [9E9, 9E9, 9E9, 9E9, 9E9, 9E9]];
	VAR jointtarget SDP_951 := [[-6.27, 35.71, 6.3, 0, 47.99, -289.51], [9E9, 9E9, 9E9, 9E9, 9E9, 9E9]];
	VAR jointtarget SDP_952 := [[-6.4, 35.76, 6.21, 0, 48.03, -289.64], [9E9, 9E9, 9E9, 9E9, 9E9, 9E9]];
	VAR jointtarget SDP_953 := [[-6.53, 35.81, 6.13, 0, 48.06, -289.77], [9E9, 9E9, 9E9, 9E9, 9E9, 9E9]];
	VAR jointtarget SDP_954 := [[-6.66, 35.86, 6.04, 0, 48.1, -289.9], [9E9, 9E9, 9E9, 9E9, 9E9, 9E9]];
	VAR jointtarget SDP_955 := [[-6.78, 35.91, 5.96, 0, 48.13, -290.02], [9E9, 9E9, 9E9, 9E9, 9E9, 9E9]];
	VAR jointtarget SDP_956 := [[-6.91, 35.96, 5.87, 0, 48.17, -290.15], [9E9, 9E9, 9E9, 9E9, 9E9, 9E9]];
	VAR jointtarget SDP_957 := [[-7.04, 36.01, 5.78, 0, 48.2, -290.28], [9E9, 9E9, 9E9, 9E9, 9E9, 9E9]];
	VAR jointtarget SDP_958 := [[-7.16, 36.06, 5.7, 0, 48.24, -290.4], [9E9, 9E9, 9E9, 9E9, 9E9, 9E9]];
	VAR jointtarget SDP_959 := [[-7.29, 36.11, 5.61, 0, 48.28, -290.53], [9E9, 9E9, 9E9, 9E9, 9E9, 9E9]];
	VAR jointtarget SDP_960 := [[-7.55, 36.17, 5.52, 0, 48.31, -280.46], [9E9, 9E9, 9E9, 9E9, 9E9, 9E9]];
	VAR jointtarget SDP_961 := [[-7.8, 36.12, 5.61, 0, 48.28, -260.07], [9E9, 9E9, 9E9, 9E9, 9E9, 9E9]];
	VAR jointtarget SDP_962 := [[-8.03, 35.97, 5.85, 0, 48.17, -239.65], [9E9, 9E9, 9E9, 9E9, 9E9, 9E9]];
	VAR jointtarget SDP_963 := [[-8.2, 35.75, 6.23, 0, 48.02, -219.17], [9E9, 9E9, 9E9, 9E9, 9E9, 9E9]];
	VAR jointtarget SDP_964 := [[-8.28, 35.48, 6.69, 0, 47.83, -198.6], [9E9, 9E9, 9E9, 9E9, 9E9, 9E9]];
	VAR jointtarget SDP_965 := [[-8.27, 35.2, 7.17, 0, 47.63, -177.95], [9E9, 9E9, 9E9, 9E9, 9E9, 9E9]];
	VAR jointtarget SDP_966 := [[-8.17, 34.94, 7.61, 0, 47.44, -157.19], [9E9, 9E9, 9E9, 9E9, 9E9, 9E9]];
	VAR jointtarget SDP_967 := [[-7.98, 34.74, 7.96, 0, 47.3, -136.36], [9E9, 9E9, 9E9, 9E9, 9E9, 9E9]];
	VAR jointtarget SDP_968 := [[-7.74, 34.62, 8.17, 0, 47.22, -115.47], [9E9, 9E9, 9E9, 9E9, 9E9, 9E9]];
	VAR jointtarget SDP_969 := [[-7.47, 34.59, 8.21, 0, 47.2, -94.56], [9E9, 9E9, 9E9, 9E9, 9E9, 9E9]];
	VAR jointtarget SDP_970 := [[-7.34, 34.61, 8.18, 0, 47.21, -84.1], [9E9, 9E9, 9E9, 9E9, 9E9, 9E9]];
	VAR jointtarget SDP_971 := [[-7.2, 34.62, 8.16, 0, 47.22, -83.96], [9E9, 9E9, 9E9, 9E9, 9E9, 9E9]];
	VAR jointtarget SDP_972 := [[-7.06, 34.63, 8.13, 0, 47.24, -83.82], [9E9, 9E9, 9E9, 9E9, 9E9, 9E9]];
	VAR jointtarget SDP_973 := [[-6.92, 34.65, 8.1, 0, 47.25, -83.68], [9E9, 9E9, 9E9, 9E9, 9E9, 9E9]];
	VAR jointtarget SDP_974 := [[-6.79, 34.66, 8.08, 0, 47.26, -83.55], [9E9, 9E9, 9E9, 9E9, 9E9, 9E9]];
	VAR jointtarget SDP_975 := [[-6.65, 34.68, 8.05, 0, 47.27, -83.41], [9E9, 9E9, 9E9, 9E9, 9E9, 9E9]];
	VAR jointtarget SDP_976 := [[-6.51, 34.7, 8.02, 0, 47.29, -83.27], [9E9, 9E9, 9E9, 9E9, 9E9, 9E9]];
	VAR jointtarget SDP_977 := [[-6.38, 34.71, 7.99, 0, 47.3, -83.14], [9E9, 9E9, 9E9, 9E9, 9E9, 9E9]];
	VAR jointtarget SDP_978 := [[-6.24, 34.73, 7.96, 0, 47.31, -83], [9E9, 9E9, 9E9, 9E9, 9E9, 9E9]];
	VAR jointtarget SDP_979 := [[-6.1, 34.74, 7.93, 0, 47.33, -82.86], [9E9, 9E9, 9E9, 9E9, 9E9, 9E9]];
	VAR jointtarget SDP_980 := [[-6.07, 34.75, 7.92, 0, 47.33, -83.49], [9E9, 9E9, 9E9, 9E9, 9E9, 9E9]];
	VAR jointtarget SDP_981 := [[-6.03, 34.75, 7.92, 0, 47.33, -84.78], [9E9, 9E9, 9E9, 9E9, 9E9, 9E9]];
	VAR jointtarget SDP_982 := [[-6, 34.75, 7.91, 0, 47.34, -86.07], [9E9, 9E9, 9E9, 9E9, 9E9, 9E9]];
	VAR jointtarget SDP_983 := [[-5.97, 34.75, 7.91, 0, 47.34, -87.36], [9E9, 9E9, 9E9, 9E9, 9E9, 9E9]];
	VAR jointtarget SDP_984 := [[-5.93, 34.76, 7.91, 0, 47.34, -88.65], [9E9, 9E9, 9E9, 9E9, 9E9, 9E9]];
